C05487=1132.913,-86.314,-45.873,178.764,6.137,149.471
C05488=1132.907,-86.064,-45.883,178.766,6.138,149.470
C05489=1132.902,-85.815,-45.892,178.768,6.139,149.470
C05490=1132.896,-85.565,-45.902,178.770,6.139,149.469
C05491=1132.891,-85.315,-45.912,178.772,6.139,149.469
C05492=1132.886,-85.064,-45.921,178.774,6.140,149.468
C05493=1132.881,-84.815,-45.931,178.777,6.140,149.468
C05494=1132.875,-84.565,-45.940,178.778,6.140,149.467
C05495=1132.871,-84.316,-45.950,178.780,6.141,149.467
C05496=1132.865,-84.066,-45.960,178.783,6.142,149.466
C05497=1132.860,-83.816,-45.969,178.785,6.143,149.466
C05498=1132.854,-83.566,-45.979,178.786,6.143,149.465
C05499=1132.849,-83.317,-45.988,178.789,6.143,149.465
C05500=1132.843,-83.067,-45.998,178.791,6.144,149.464
C05501=1132.838,-82.818,-46.007,178.793,6.144,149.464
C05502=1132.833,-82.567,-46.018,178.795,6.144,149.463
C05503=1132.828,-82.318,-46.027,178.797,6.145,149.463
C05504=1132.822,-82.068,-46.037,178.799,6.146,149.462
C05505=1132.817,-81.818,-46.046,178.802,6.147,149.462
C05506=1132.812,-81.569,-46.056,178.804,6.146,149.461
C05507=1132.806,-81.318,-46.066,178.806,6.147,149.461
C05508=1132.801,-81.069,-46.075,178.808,6.148,149.460
C05509=1132.795,-80.820,-46.086,178.810,6.149,149.460
C05510=1132.791,-80.569,-46.095,178.812,6.148,149.459
C05511=1132.785,-80.320,-46.105,178.814,6.149,149.459
C05512=1132.779,-80.069,-46.114,178.816,6.150,149.458
C05513=1132.774,-79.820,-46.124,178.819,6.150,149.457
C05514=1132.769,-79.571,-46.134,178.821,6.150,149.457
C05515=1132.764,-79.321,-46.143,178.823,6.151,149.456
C05516=1132.758,-79.071,-46.153,178.825,6.152,149.456
C05517=1132.753,-78.821,-46.164,178.827,6.153,149.456
C05518=1132.748,-78.571,-46.173,178.829,6.153,149.455
C05519=1132.742,-78.322,-46.183,178.831,6.153,149.455
C05520=1132.737,-78.072,-46.193,178.834,6.154,149.454
C05521=1132.732,-77.822,-46.202,178.836,6.154,149.453
C05522=1132.726,-77.573,-46.212,178.837,6.154,149.453
C05523=1132.721,-77.301,-46.223,178.840,6.155,149.452
C05524=1132.715,-77.029,-46.234,178.842,6.156,149.452
C05525=1132.709,-76.759,-46.245,178.844,6.156,149.451
C05526=1132.703,-76.487,-46.255,178.847,6.157,149.451
C05527=1132.698,-76.237,-46.265,178.849,6.158,149.450
C05528=1132.693,-75.987,-46.276,178.852,6.158,149.450
C05529=1132.687,-75.737,-46.285,178.853,6.158,149.449
C05530=1132.682,-75.487,-46.295,178.855,6.159,149.449
C05531=1132.676,-75.238,-46.305,178.858,6.160,149.448
C05532=1132.671,-74.988,-46.315,178.860,6.160,149.448
C05533=1132.666,-74.738,-46.325,178.862,6.161,149.447
C05534=1132.661,-74.488,-46.335,178.864,6.161,149.446
C05535=1132.655,-74.239,-46.345,178.866,6.162,149.446
C05536=1132.649,-73.989,-46.355,178.868,6.162,149.445
C05537=1132.644,-73.739,-46.364,178.871,6.163,149.445
C05538=1132.639,-73.489,-46.375,178.872,6.163,149.444
C05539=1132.634,-73.240,-46.385,178.874,6.164,149.444
C05540=1132.628,-72.990,-46.395,178.877,6.164,149.443
C05541=1132.623,-72.741,-46.405,178.879,6.165,149.443
C05542=1132.618,-72.490,-46.415,178.881,6.166,149.442
C05543=1132.612,-72.240,-46.425,178.883,6.166,149.442
C05544=1132.607,-71.991,-46.435,178.885,6.166,149.441
C05545=1132.602,-71.742,-46.445,178.888,6.167,149.441
C05546=1132.597,-71.491,-46.455,178.890,6.167,149.440
C05547=1132.591,-71.242,-46.465,178.892,6.168,149.440
C05548=1132.586,-70.992,-46.476,178.894,6.168,149.439
C05549=1132.581,-70.743,-46.485,178.896,6.169,149.439
C05550=1132.576,-70.493,-46.496,178.898,6.170,149.438
C05551=1132.570,-70.243,-46.505,178.901,6.170,149.438
C05552=1132.564,-69.993,-46.515,178.903,6.171,149.437
C05553=1132.559,-69.743,-46.526,178.905,6.171,149.437
C05554=1132.554,-69.493,-46.536,178.907,6.172,149.436
C05555=1132.549,-69.244,-46.546,178.909,6.172,149.436
C05556=1132.543,-68.994,-46.556,178.912,6.173,149.435
C05557=1132.538,-68.744,-46.567,178.914,6.173,149.434
C05558=1132.533,-68.495,-46.577,178.916,6.174,149.434
C05559=1132.527,-68.245,-46.587,178.918,6.174,149.433
C05560=1132.522,-67.995,-46.598,178.920,6.175,149.433
C05561=1132.517,-67.746,-46.607,178.923,6.175,149.432
C05562=1132.511,-67.496,-46.617,178.925,6.176,149.432
C05563=1132.506,-67.246,-46.628,178.927,6.177,149.431
C05564=1132.501,-66.996,-46.638,178.929,6.177,149.431
C05565=1132.495,-66.747,-46.648,178.931,6.178,149.430
C05566=1132.490,-66.497,-46.659,178.933,6.178,149.430
C05567=1132.485,-66.247,-46.669,178.936,6.179,149.429
C05568=1132.480,-65.998,-46.679,178.938,6.180,149.429
C05569=1132.475,-65.748,-46.689,178.940,6.180,149.428
C05570=1132.469,-65.498,-46.700,178.942,6.180,149.428
C05571=1132.464,-65.248,-46.710,178.944,6.181,149.427
C05572=1132.459,-64.998,-46.720,178.946,6.181,149.426
C05573=1132.453,-64.749,-46.731,178.949,6.182,149.426
C05574=1132.447,-64.499,-46.741,178.951,6.183,149.426
C05575=1132.442,-64.249,-46.751,178.953,6.184,149.425
C05576=1132.437,-63.999,-46.762,178.955,6.184,149.425
C05577=1132.432,-63.749,-46.772,178.957,6.184,149.424
C05578=1132.426,-63.500,-46.782,178.959,6.185,149.423
C05579=1132.422,-63.251,-46.793,178.962,6.186,149.423
C05580=1132.417,-63.001,-46.803,178.964,6.186,149.422
C05581=1132.411,-62.751,-46.813,178.967,6.187,149.422
C05582=1132.406,-62.502,-46.824,178.969,6.187,149.421
C05583=1132.401,-62.251,-46.834,178.970,6.187,149.421
C05584=1132.395,-62.002,-46.844,178.973,6.188,149.420
C05585=1132.390,-61.752,-46.855,178.975,6.189,149.420
C05586=1132.385,-61.503,-46.866,178.977,6.189,149.419
C05587=1132.380,-61.252,-46.877,178.980,6.190,149.419
C05588=1132.374,-61.003,-46.887,178.982,6.191,149.418
C05589=1132.368,-60.753,-46.897,178.984,6.192,149.418
C05590=1132.363,-60.503,-46.908,178.986,6.192,149.417
C05591=1132.358,-60.254,-46.918,178.988,6.192,149.416
C05592=1132.353,-60.004,-46.929,178.990,6.193,149.416
C05593=1132.348,-59.754,-46.939,178.993,6.194,149.415
C05594=1132.343,-59.504,-46.950,178.995,6.194,149.415
C05595=1132.337,-59.255,-46.960,178.997,6.195,149.414
C05596=1132.331,-59.005,-46.970,179.000,6.195,149.414
C05597=1132.327,-58.755,-46.982,179.002,6.196,149.413
C05598=1132.321,-58.506,-46.992,179.003,6.196,149.413
C05599=1132.316,-58.256,-47.002,179.006,6.197,149.412
C05600=1132.310,-58.006,-47.013,179.008,6.197,149.412
C05601=1132.306,-57.756,-47.024,179.010,6.198,149.411
C05602=1132.300,-57.507,-47.034,179.013,6.199,149.411
C05603=1132.294,-57.256,-47.045,179.015,6.200,149.410
C05604=1132.289,-57.007,-47.056,179.018,6.200,149.410
C05605=1132.284,-56.757,-47.067,179.020,6.201,149.409
C05606=1132.279,-56.508,-47.077,179.021,6.201,149.409
C05607=1132.274,-56.258,-47.088,179.024,6.202,149.408
C05608=1132.268,-56.008,-47.098,179.026,6.202,149.408
C05609=1132.263,-55.758,-47.109,179.028,6.203,149.407
C05610=1132.258,-55.509,-47.120,179.031,6.203,149.406
C05611=1132.253,-55.259,-47.130,179.033,6.204,149.406
C05612=1132.247,-55.009,-47.141,179.035,6.205,149.405
C05613=1132.243,-54.760,-47.152,179.038,6.205,149.405
C05614=1132.237,-54.510,-47.162,179.040,6.206,149.404
C05615=1132.231,-54.260,-47.173,179.042,6.207,149.404
C05616=1132.226,-54.011,-47.184,179.044,6.207,149.403
C05617=1132.221,-53.761,-47.195,179.046,6.208,149.403
C05618=1132.215,-53.511,-47.205,179.048,6.208,149.402
C05619=1132.211,-53.261,-47.216,179.051,6.209,149.402
C05620=1132.205,-53.012,-47.227,179.053,6.210,149.401
C05621=1132.200,-52.762,-47.238,179.055,6.210,149.401
C05622=1132.194,-52.512,-47.249,179.058,6.211,149.400
C05623=1132.189,-52.263,-47.260,179.060,6.211,149.400
C05624=1132.184,-52.013,-47.270,179.062,6.212,149.399
C05625=1132.179,-51.763,-47.281,179.064,6.213,149.399
C05626=1132.174,-51.514,-47.292,179.067,6.213,149.398
C05627=1132.168,-51.243,-47.304,179.069,6.214,149.397
C05628=1132.162,-50.971,-47.315,179.071,6.215,149.397
C05629=1132.156,-50.701,-47.327,179.074,6.215,149.396
C05630=1132.151,-50.431,-47.339,179.076,6.216,149.396
C05631=1132.145,-50.180,-47.350,179.079,6.216,149.395
C05632=1132.140,-49.931,-47.361,179.081,6.217,149.395
C05633=1132.135,-49.681,-47.372,179.083,6.218,149.394
C05634=1132.130,-49.432,-47.383,179.085,6.219,149.394
C05635=1132.124,-49.181,-47.394,179.088,6.219,149.393
C05636=1132.119,-48.932,-47.405,179.090,6.219,149.392
C05637=1132.114,-48.683,-47.416,179.092,6.220,149.392
C05638=1132.109,-48.433,-47.427,179.094,6.221,149.391
C05639=1132.103,-48.183,-47.438,179.097,6.221,149.391
C05640=1132.098,-47.933,-47.449,179.099,6.222,149.390
C05641=1132.093,-47.684,-47.460,179.101,6.223,149.390
C05642=1132.088,-47.434,-47.470,179.103,6.223,149.389
C05643=1132.082,-47.184,-47.482,179.106,6.224,149.389
C05644=1132.077,-46.935,-47.493,179.108,6.225,149.388
C05645=1132.072,-46.685,-47.504,179.110,6.225,149.388
C05646=1132.066,-46.435,-47.515,179.113,6.226,149.387
C05647=1132.061,-46.185,-47.526,179.115,6.226,149.386
C05648=1132.056,-45.936,-47.537,179.117,6.227,149.386
C05649=1132.050,-45.686,-47.548,179.120,6.228,149.386
C05650=1132.045,-45.436,-47.559,179.122,6.229,149.385
C05651=1132.040,-45.187,-47.570,179.124,6.229,149.384
C05652=1132.034,-44.937,-47.582,179.127,6.230,149.384
C05653=1132.029,-44.687,-47.592,179.129,6.231,149.383
C05654=1132.025,-44.437,-47.604,179.131,6.231,149.383
C05655=1132.019,-44.188,-47.615,179.134,6.232,149.382
C05656=1132.014,-43.938,-47.626,179.135,6.232,149.382
C05657=1132.009,-43.688,-47.637,179.137,6.233,149.381
C05658=1132.003,-43.439,-47.649,179.140,6.233,149.381
C05659=1131.998,-43.189,-47.659,179.142,6.234,149.380
C05660=1131.993,-42.939,-47.671,179.144,6.235,149.380
C05661=1131.987,-42.690,-47.682,179.147,6.235,149.379
C05662=1131.983,-42.440,-47.693,179.149,6.236,149.379
C05663=1131.977,-42.190,-47.704,179.152,6.236,149.378
C05664=1131.972,-41.941,-47.715,179.154,6.237,149.377
C05665=1131.967,-41.691,-47.727,179.156,6.238,149.377
C05666=1131.961,-41.441,-47.739,179.159,6.238,149.376
C05667=1131.956,-41.191,-47.749,179.161,6.239,149.376
C05668=1131.950,-40.942,-47.761,179.163,6.240,149.375
C05669=1131.946,-40.692,-47.772,179.165,6.241,149.375
C05670=1131.940,-40.442,-47.784,179.168,6.241,149.374
C05671=1131.935,-40.193,-47.794,179.170,6.242,149.374
C05672=1131.929,-39.943,-47.806,179.172,6.243,149.373
C05673=1131.925,-39.693,-47.817,179.174,6.243,149.373
C05674=1131.920,-39.444,-47.828,179.177,6.244,149.372
C05675=1131.914,-39.194,-47.840,179.179,6.245,149.372
C05676=1131.909,-38.945,-47.851,179.181,6.245,149.371
C05677=1131.903,-38.694,-47.862,179.184,6.246,149.371
C05678=1131.898,-38.445,-47.873,179.186,6.247,149.370
C05679=1131.893,-38.195,-47.885,179.188,6.247,149.369
C05680=1131.888,-37.946,-47.897,179.191,6.248,149.369
C05681=1131.883,-37.696,-47.908,179.193,6.248,149.368
C05682=1131.877,-37.447,-47.919,179.195,6.249,149.368
C05683=1131.872,-37.197,-47.931,179.198,6.250,149.367
C05684=1131.867,-36.947,-47.943,179.200,6.251,149.367
C05685=1131.861,-36.697,-47.954,179.203,6.251,149.366
C05686=1131.856,-36.447,-47.966,179.205,6.252,149.366
C05687=1131.851,-36.198,-47.976,179.207,6.253,149.365
C05688=1131.845,-35.948,-47.988,179.209,6.254,149.365
C05689=1131.841,-35.698,-48.000,179.212,6.254,149.364
C05690=1131.835,-35.448,-48.012,179.214,6.255,149.363
C05691=1131.830,-35.199,-48.022,179.216,6.256,149.363
C05692=1131.824,-34.949,-48.034,179.219,6.256,149.362
C05693=1131.820,-34.700,-48.046,179.221,6.257,149.362
C05694=1131.814,-34.450,-48.058,179.223,6.257,149.361
C05695=1131.809,-34.200,-48.069,179.225,6.258,149.361
C05696=1131.804,-33.951,-48.080,179.228,6.259,149.360
C05697=1131.798,-33.701,-48.092,179.230,6.259,149.360
C05698=1131.793,-33.451,-48.104,179.232,6.260,149.359
C05699=1131.788,-33.202,-48.115,179.235,6.261,149.359
C05700=1131.783,-32.952,-48.127,179.237,6.261,149.358
C05701=1131.778,-32.702,-48.139,179.239,6.262,149.358
C05702=1131.772,-32.453,-48.150,179.242,6.263,149.357
C05703=1131.767,-32.203,-48.161,179.245,6.264,149.356
C05704=1131.762,-31.953,-48.173,179.247,6.265,149.356
C05705=1131.756,-31.703,-48.185,179.249,6.266,149.355
C05706=1131.752,-31.454,-48.196,179.251,6.266,149.355
C05707=1131.746,-31.204,-48.209,179.254,6.267,149.354
C05708=1131.741,-30.954,-48.221,179.256,6.268,149.354
C05709=1131.736,-30.705,-48.232,179.258,6.268,149.353
C05710=1131.730,-30.456,-48.244,179.261,6.269,149.353
C05711=1131.725,-30.206,-48.256,179.263,6.270,149.352
C05712=1131.720,-29.956,-48.267,179.266,6.270,149.352
C05713=1131.715,-29.706,-48.279,179.268,6.271,149.351
C05714=1131.709,-29.456,-48.291,179.270,6.272,149.351
C05715=1131.705,-29.207,-48.303,179.273,6.272,149.350
C05716=1131.700,-28.957,-48.315,179.275,6.273,149.350
C05717=1131.693,-28.708,-48.326,179.277,6.273,149.349
C05718=1131.689,-28.458,-48.337,179.280,6.274,149.348
C05719=1131.683,-28.208,-48.349,179.282,6.275,149.348
C05720=1131.678,-27.958,-48.361,179.284,6.275,149.347
C05721=1131.673,-27.709,-48.374,179.287,6.276,149.347
C05722=1131.668,-27.459,-48.385,179.289,6.278,149.346
C05723=1131.663,-27.210,-48.397,179.292,6.279,149.346
C05724=1131.657,-26.960,-48.409,179.294,6.279,149.345
C05725=1131.653,-26.711,-48.421,179.296,6.280,149.345
C05726=1131.647,-26.461,-48.433,179.299,6.281,149.344
C05727=1131.642,-26.211,-48.445,179.301,6.281,149.343
C05728=1131.637,-25.961,-48.456,179.303,6.282,149.343
C05729=1131.632,-25.712,-48.468,179.306,6.283,149.343
C05730=1131.627,-25.462,-48.480,179.308,6.283,149.342
C05731=1131.621,-25.192,-48.493,179.311,6.284,149.341
C05732=1131.615,-24.922,-48.507,179.313,6.285,149.341
C05733=1131.609,-24.652,-48.519,179.316,6.286,149.340
C05734=1131.604,-24.382,-48.532,179.318,6.286,149.340
C05735=1131.598,-24.132,-48.544,179.321,6.287,149.339
C05736=1131.594,-23.883,-48.556,179.323,6.288,149.339
C05737=1131.588,-23.633,-48.568,179.325,6.288,149.338
C05738=1131.583,-23.383,-48.580,179.328,6.290,149.337
C05739=1131.578,-23.133,-48.592,179.331,6.290,149.337
C05740=1131.572,-22.883,-48.604,179.333,6.291,149.336
C05741=1131.567,-22.633,-48.616,179.335,6.292,149.336
C05742=1131.562,-22.384,-48.629,179.338,6.292,149.335
C05743=1131.557,-22.135,-48.640,179.340,6.293,149.335
C05744=1131.552,-21.885,-48.652,179.342,6.294,149.334
C05745=1131.547,-21.635,-48.665,179.345,6.294,149.334
C05746=1131.541,-21.385,-48.676,179.347,6.295,149.333
C05747=1131.536,-21.136,-48.689,179.349,6.296,149.333
C05748=1131.531,-20.886,-48.701,179.352,6.297,149.332
C05749=1131.525,-20.636,-48.713,179.355,6.298,149.331
C05750=1131.520,-20.387,-48.725,179.357,6.299,149.331
C05751=1131.515,-20.137,-48.737,179.359,6.299,149.331
C05752=1131.510,-19.888,-48.749,179.362,6.300,149.330
C05753=1131.505,-19.638,-48.761,179.364,6.301,149.329
C05754=1131.500,-19.389,-48.774,179.366,6.301,149.329
C05755=1131.494,-19.139,-48.786,179.369,6.302,149.328
C05756=1131.489,-18.889,-48.798,179.371,6.303,149.328
C05757=1131.484,-18.639,-48.810,179.374,6.304,149.327
C05758=1131.479,-18.390,-48.823,179.376,6.305,149.327
C05759=1131.473,-18.140,-48.835,179.378,6.305,149.326
C05760=1131.468,-17.891,-48.847,179.381,6.306,149.326
C05761=1131.463,-17.641,-48.859,179.383,6.307,149.325
C05762=1131.457,-17.392,-48.872,179.385,6.307,149.324
C05763=1131.453,-17.141,-48.884,179.388,6.308,149.324
C05764=1131.447,-16.892,-48.897,179.390,6.310,149.324
C05765=1131.442,-16.642,-48.909,179.393,6.310,149.323
C05766=1131.437,-16.392,-48.921,179.395,6.311,149.322
C05767=1131.432,-16.143,-48.934,179.397,6.312,149.322
C05768=1131.426,-15.893,-48.946,179.400,6.312,149.321
C05769=1131.421,-15.644,-48.958,179.402,6.313,149.321
C05770=1131.416,-15.394,-48.970,179.404,6.314,149.320
C05771=1131.411,-15.145,-48.983,179.407,6.315,149.320
C05772=1131.406,-14.895,-48.995,179.410,6.316,149.319
C05773=1131.401,-14.645,-49.007,179.412,6.316,149.319
C05774=1131.396,-14.395,-49.020,179.414,6.317,149.318
C05775=1131.391,-14.146,-49.033,179.417,6.318,149.317
C05776=1131.385,-13.896,-49.045,179.419,6.318,149.317
C05777=1131.380,-13.647,-49.057,179.421,6.319,149.317
C05778=1131.375,-13.397,-49.070,179.425,6.320,149.316
C05779=1131.369,-13.148,-49.082,179.427,6.321,149.315
C05780=1131.364,-12.898,-49.094,179.429,6.322,149.315
C05781=1131.360,-12.648,-49.107,179.431,6.323,149.314
C05782=1131.354,-12.398,-49.119,179.434,6.323,149.314
C05783=1131.348,-12.149,-49.132,179.436,6.324,149.313
C05784=1131.343,-11.899,-49.145,179.439,6.326,149.313
C05785=1131.338,-11.650,-49.157,179.441,6.326,149.312
C05786=1131.333,-11.400,-49.169,179.444,6.327,149.312
C05787=1131.328,-11.150,-49.182,179.446,6.328,149.311
C05788=1131.323,-10.901,-49.195,179.448,6.328,149.310
C05789=1131.318,-10.651,-49.208,179.451,6.330,149.310
C05790=1131.313,-10.401,-49.219,179.453,6.330,149.310
C05791=1131.307,-10.152,-49.232,179.456,6.331,149.309
C05792=1131.302,-9.902,-49.246,179.458,6.332,149.308
C05793=1131.297,-9.652,-49.258,179.460,6.332,149.308
C05794=1131.292,-9.403,-49.271,179.463,6.333,149.307
C05795=1131.287,-9.153,-49.283,179.466,6.334,149.307
C05796=1131.281,-8.904,-49.295,179.468,6.335,149.306
C05797=1131.277,-8.654,-49.308,179.470,6.336,149.306
C05798=1131.271,-8.404,-49.321,179.473,6.336,149.305
C05799=1131.266,-8.155,-49.334,179.475,6.337,149.305
C05800=1131.261,-7.906,-49.347,179.478,6.339,149.304
C05801=1131.256,-7.655,-49.359,179.480,6.339,149.303
C05802=1131.251,-7.406,-49.371,179.483,6.340,149.303
C05803=1131.245,-7.156,-49.385,179.485,6.341,149.303
C05804=1131.240,-6.907,-49.397,179.487,6.341,149.302
C05805=1131.235,-6.657,-49.410,179.490,6.343,149.301
C05806=1131.230,-6.407,-49.423,179.492,6.344,149.301
C05807=1131.225,-6.158,-49.435,179.495,6.344,149.300
C05808=1131.219,-5.908,-49.449,179.497,6.345,149.300
C05809=1131.215,-5.658,-49.462,179.499,6.346,149.299
C05810=1131.210,-5.409,-49.474,179.502,6.347,149.299
C05811=1131.204,-5.160,-49.487,179.505,6.348,149.298
C05812=1131.199,-4.910,-49.500,179.507,6.348,149.298
C05813=1131.194,-4.660,-49.513,179.509,6.349,149.297
C05814=1131.189,-4.411,-49.526,179.512,6.350,149.296
C05815=1131.183,-4.161,-49.539,179.515,6.351,149.296
C05816=1131.179,-3.911,-49.552,179.517,6.352,149.296
C05817=1131.173,-3.662,-49.564,179.520,6.352,149.295
C05818=1131.168,-3.413,-49.577,179.522,6.353,149.294
C05819=1131.162,-3.163,-49.590,179.525,6.355,149.294
C05820=1131.158,-2.913,-49.603,179.527,6.355,149.293
C05821=1131.153,-2.664,-49.616,179.529,6.356,149.293
C05822=1131.147,-2.414,-49.629,179.532,6.357,149.292
C05823=1131.142,-2.164,-49.642,179.534,6.358,149.292
C05824=1131.137,-1.915,-49.654,179.537,6.359,149.291
C05825=1131.131,-1.665,-49.668,179.539,6.360,149.291
C05826=1131.127,-1.415,-49.681,179.541,6.360,149.290
C05827=1131.122,-1.166,-49.693,179.545,6.362,149.290
C05828=1131.116,-0.916,-49.706,179.547,6.362,149.289
C05829=1131.111,-0.666,-49.719,179.549,6.363,149.289
C05830=1131.106,-0.416,-49.733,179.552,6.364,149.288
C05831=1131.101,-0.168,-49.746,179.554,6.364,149.287
C05832=1131.096,0.082,-49.759,179.557,6.366,149.287
C05833=1131.090,0.332,-49.772,179.559,6.366,149.286
C05834=1131.085,0.581,-49.785,179.561,6.367,149.286
C05835=1131.079,0.851,-49.799,179.564,6.369,149.285
C05836=1131.075,1.120,-49.813,179.567,6.369,149.285
C05837=1131.068,1.390,-49.827,179.570,6.371,149.284
C05838=1131.063,1.660,-49.842,179.572,6.371,149.284
C05839=1131.058,1.910,-49.854,179.574,6.372,149.283
C05840=1131.053,2.159,-49.868,179.578,6.373,149.282
C05841=1131.047,2.408,-49.881,179.580,6.374,149.282
C05842=1131.043,2.658,-49.894,179.582,6.375,149.281
C05843=1131.037,2.908,-49.907,179.584,6.376,149.281
C05844=1131.033,3.158,-49.920,179.587,6.377,149.280
C05845=1131.027,3.407,-49.934,179.590,6.378,149.280
C05846=1131.022,3.656,-49.947,179.592,6.378,149.279
C05847=1131.017,3.906,-49.960,179.594,6.379,149.279
C05848=1131.012,4.155,-49.974,179.597,6.380,149.278
C05849=1131.007,4.406,-49.987,179.599,6.381,149.278
C05850=1131.001,4.655,-50.000,179.602,6.382,149.277
C05851=1130.996,4.905,-50.013,179.605,6.383,149.277
C05852=1130.991,5.154,-50.027,179.607,6.384,149.276
C05853=1130.985,5.403,-50.040,179.610,6.384,149.275
C05854=1130.981,5.653,-50.053,179.612,6.385,149.275
C05855=1130.975,5.902,-50.067,179.615,6.387,149.274
C05856=1130.971,6.153,-50.080,179.617,6.387,149.274
C05857=1130.965,6.402,-50.093,179.620,6.388,149.273
C05858=1130.960,6.652,-50.107,179.622,6.390,149.273
C05859=1130.955,6.901,-50.120,179.624,6.391,149.272
C05860=1130.950,7.151,-50.134,179.627,6.391,149.272
C05861=1130.945,7.400,-50.147,179.629,6.392,149.271
C05862=1130.940,7.651,-50.160,179.632,6.393,149.271
C05863=1130.935,7.899,-50.173,179.635,6.394,149.270
C05864=1130.930,8.150,-50.187,179.637,6.395,149.270
C05865=1130.924,8.399,-50.201,179.640,6.396,149.269
C05866=1130.919,8.649,-50.214,179.642,6.397,149.268
C05867=1130.914,8.898,-50.228,179.645,6.397,149.268
C05868=1130.909,9.148,-50.241,179.647,6.399,149.268
C05869=1130.904,9.397,-50.254,179.650,6.399,149.267
C05870=1130.899,9.647,-50.268,179.652,6.400,149.266
C05871=1130.893,9.896,-50.281,179.655,6.402,149.266
C05872=1130.888,10.146,-50.295,179.658,6.402,149.265
C05873=1130.883,10.396,-50.308,179.660,6.403,149.265
C05874=1130.878,10.645,-50.322,179.662,6.405,149.264
C05875=1130.873,10.895,-50.335,179.665,6.405,149.264
C05876=1130.868,11.144,-50.349,179.667,6.406,149.263
C05877=1130.862,11.394,-50.362,179.670,6.407,149.263
C05878=1130.858,11.643,-50.376,179.672,6.408,149.262
C05879=1130.853,11.893,-50.391,179.675,6.409,149.262
C05880=1130.847,12.142,-50.403,179.678,6.410,149.261
C05881=1130.842,12.392,-50.417,179.680,6.411,149.261
C05882=1130.837,12.642,-50.431,179.683,6.412,149.260
C05883=1130.832,12.891,-50.444,179.685,6.413,149.260
C05884=1130.827,13.141,-50.458,179.687,6.414,149.259
C05885=1130.822,13.390,-50.472,179.690,6.414,149.258
C05886=1130.817,13.640,-50.486,179.693,6.416,149.258
C05887=1130.811,13.890,-50.499,179.695,6.417,149.257
C05888=1130.807,14.139,-50.513,179.697,6.418,149.257
C05889=1130.801,14.388,-50.527,179.701,6.419,149.256
C05890=1130.796,14.639,-50.540,179.703,6.420,149.256
C05891=1130.792,14.888,-50.554,179.705,6.420,149.255
C05892=1130.786,15.137,-50.568,179.708,6.422,149.255
C05893=1130.781,15.387,-50.582,179.710,6.422,149.254
C05894=1130.775,15.636,-50.596,179.712,6.423,149.254
C05895=1130.771,15.886,-50.609,179.716,6.424,149.253
C05896=1130.766,16.136,-50.623,179.718,6.425,149.253
C05897=1130.760,16.385,-50.637,179.720,6.426,149.252
C05898=1130.755,16.635,-50.651,179.723,6.427,149.251
C05899=1130.750,16.884,-50.665,179.725,6.428,149.251
C05900=1130.745,17.134,-50.678,179.728,6.430,149.251
C05901=1130.740,17.384,-50.692,179.731,6.430,149.250
C05902=1130.735,17.633,-50.706,179.733,6.431,149.249
C05903=1130.730,17.882,-50.720,179.736,6.433,149.249
C05904=1130.724,18.133,-50.734,179.738,6.433,149.249
C05905=1130.719,18.382,-50.748,179.741,6.434,149.248
C05906=1130.715,18.631,-50.761,179.743,6.435,149.247
C05907=1130.710,18.881,-50.776,179.746,6.436,149.247
C05908=1130.704,19.130,-50.790,179.749,6.437,149.246
C05909=1130.699,19.380,-50.803,179.751,6.438,149.246
C05910=1130.694,19.630,-50.817,179.753,6.439,149.245
C05911=1130.689,19.879,-50.832,179.756,6.440,149.245
C05912=1130.683,20.128,-50.846,179.759,6.441,149.244
C05913=1130.678,20.378,-50.860,179.761,6.443,149.244
C05914=1130.673,20.628,-50.874,179.764,6.444,149.243
C05915=1130.669,20.877,-50.888,179.766,6.444,149.243
C05916=1130.663,21.127,-50.901,179.769,6.446,149.242
C05917=1130.658,21.377,-50.915,179.771,6.446,149.242
C05918=1130.653,21.626,-50.930,179.774,6.448,149.241
C05919=1130.648,21.875,-50.944,179.777,6.448,149.241
C05920=1130.643,22.125,-50.958,179.779,6.449,149.240
C05921=1130.638,22.375,-50.972,179.782,6.450,149.239
C05922=1130.632,22.624,-50.986,179.784,6.451,149.239
C05923=1130.627,22.873,-51.000,179.787,6.453,149.238
C05924=1130.623,23.123,-51.015,179.790,6.453,149.238
C05925=1130.618,23.373,-51.029,179.792,6.454,149.237
C05926=1130.612,23.622,-51.043,179.795,6.456,149.237
C05927=1130.607,23.872,-51.057,179.797,6.457,149.236
C05928=1130.602,24.121,-51.071,179.800,6.458,149.236
C05929=1130.597,24.371,-51.086,179.802,6.459,149.235
C05930=1130.592,24.621,-51.100,179.804,6.459,149.235
C05931=1130.587,24.870,-51.114,179.808,6.461,149.234
C05932=1130.582,25.119,-51.128,179.810,6.461,149.234
C05933=1130.577,25.369,-51.142,179.813,6.463,149.233
C05934=1130.572,25.619,-51.157,179.815,6.463,149.233
C05935=1130.566,25.868,-51.171,179.818,6.465,149.232
C05936=1130.561,26.118,-51.185,179.820,6.466,149.232
C05937=1130.556,26.367,-51.199,179.822,6.467,149.231
C05938=1130.551,26.617,-51.213,179.826,6.468,149.231
C05939=1130.546,26.886,-51.229,179.828,6.470,149.230
C05940=1130.540,27.155,-51.245,179.831,6.470,149.229
C05941=1130.534,27.424,-51.260,179.834,6.472,149.229
C05942=1130.529,27.692,-51.276,179.836,6.472,149.228
C05943=1130.524,27.942,-51.290,179.839,6.474,149.228
C05944=1130.519,28.192,-51.304,179.841,6.474,149.227
C05945=1130.514,28.442,-51.319,179.845,6.476,149.227
C05946=1130.509,28.691,-51.333,179.847,6.477,149.226
C05947=1130.504,28.941,-51.348,179.850,6.478,149.226
C05948=1130.498,29.190,-51.362,179.852,6.479,149.225
C05949=1130.493,29.439,-51.377,179.855,6.480,149.225
C05950=1130.489,29.689,-51.391,179.857,6.481,149.224
C05951=1130.484,29.939,-51.405,179.860,6.483,149.224
C05952=1130.479,30.188,-51.420,179.863,6.483,149.223
C05953=1130.474,30.438,-51.434,179.865,6.484,149.223
C05954=1130.468,30.688,-51.449,179.867,6.485,149.222
C05955=1130.463,30.937,-51.464,179.870,6.486,149.222
C05956=1130.458,31.186,-51.478,179.873,6.488,149.221
C05957=1130.453,31.435,-51.492,179.875,6.488,149.221
C05958=1130.448,31.685,-51.507,179.878,6.490,149.220
C05959=1130.442,31.935,-51.522,179.880,6.490,149.219
C05960=1130.438,32.184,-51.537,179.883,6.492,149.219
C05961=1130.433,32.434,-51.551,179.885,6.493,149.218
C05962=1130.428,32.684,-51.565,179.889,6.494,149.218
C05963=1130.423,32.933,-51.580,179.891,6.495,149.217
C05964=1130.418,33.183,-51.595,179.894,6.497,149.217
C05965=1130.413,33.433,-51.609,179.896,6.497,149.216
C05966=1130.408,33.682,-51.624,179.899,6.499,149.216
C05967=1130.402,33.931,-51.638,179.901,6.499,149.215
C05968=1130.397,34.181,-51.653,179.904,6.501,149.215
C05969=1130.392,34.430,-51.668,179.907,6.501,149.214
C05970=1130.387,34.679,-51.682,179.909,6.503,149.214
C05971=1130.382,34.929,-51.698,179.912,6.504,149.213
C05972=1130.377,35.179,-51.712,179.914,6.505,149.213
C05973=1130.372,35.428,-51.727,179.917,6.506,149.212
C05974=1130.367,35.677,-51.741,179.920,6.508,149.212
C05975=1130.361,35.927,-51.756,179.922,6.508,149.211
C05976=1130.357,36.176,-51.771,179.925,6.510,149.211
C05977=1130.352,36.426,-51.786,179.927,6.510,149.210
C05978=1130.346,36.676,-51.801,179.930,6.512,149.210
C05979=1130.342,36.925,-51.815,179.932,6.513,149.209
C05980=1130.337,37.174,-51.830,179.935,6.514,149.209
C05981=1130.331,37.424,-51.845,179.938,6.515,149.208
C05982=1130.327,37.673,-51.860,179.940,6.517,149.208
C05983=1130.321,37.924,-51.875,179.943,6.517,149.207
C05984=1130.316,38.173,-51.890,179.946,6.519,149.207
C05985=1130.311,38.422,-51.904,179.948,6.519,149.206
C05986=1130.306,38.672,-51.920,179.951,6.521,149.206
C05987=1130.301,38.905,-51.934,179.953,6.522,149.205
C05988=1130.297,39.137,-51.948,179.956,6.523,149.204
C05989=1130.293,39.369,-51.962,179.958,6.524,149.204
C05990=1130.268,40.531,-52.031,179.713,7.030,149.388
C05991=1130.263,40.781,-52.047,179.714,7.034,149.388
C05992=1130.259,41.031,-52.062,179.715,7.039,149.389
C05993=1130.253,41.281,-52.077,179.716,7.043,149.390
C05994=1130.249,41.530,-52.092,179.718,7.047,149.390
C05995=1130.243,41.779,-52.108,179.719,7.052,149.391
C05996=1130.239,42.028,-52.123,179.721,7.056,149.391
C05997=1130.233,42.278,-52.138,179.722,7.060,149.392
C05998=1130.227,42.528,-52.153,179.723,7.064,149.392
C05999=1130.223,42.777,-52.168,179.724,7.069,149.393
C06000=1130.218,43.027,-52.184,179.726,7.073,149.394
C06001=1130.213,43.276,-52.199,179.727,7.077,149.394
C06002=1130.208,43.525,-52.215,179.728,7.081,149.395
C06003=1130.203,43.774,-52.230,179.729,7.085,149.395
C06004=1130.198,44.025,-52.244,179.731,7.089,149.396
C06005=1130.192,44.274,-52.260,179.732,7.093,149.396
C06006=1130.188,44.524,-52.275,179.733,7.098,149.397
C06007=1130.183,44.773,-52.291,179.734,7.102,149.398
C06008=1130.177,45.023,-52.307,179.736,7.106,149.398
C06009=1130.173,45.272,-52.322,179.737,7.110,149.399
C06010=1130.167,45.521,-52.337,179.738,7.114,149.399
C06011=1130.163,45.771,-52.353,179.740,7.118,149.400
C06012=1130.158,46.020,-52.368,179.741,7.123,149.400
C06013=1130.153,46.270,-52.384,179.742,7.127,149.401
C06014=1130.148,46.519,-52.399,179.743,7.131,149.401
C06015=1130.143,46.769,-52.415,179.745,7.135,149.402
C06016=1130.138,47.018,-52.430,179.746,7.139,149.403
C06017=1130.132,47.268,-52.446,179.747,7.143,149.403
C06018=1130.128,47.517,-52.461,179.749,7.147,149.404
C06019=1130.124,47.735,-52.475,179.750,7.151,149.404
C06020=1130.119,47.953,-52.488,179.751,7.154,149.404
C06021=1130.115,48.170,-52.501,179.752,7.159,149.405
C06022=1130.110,48.388,-52.516,179.753,7.162,149.406
C06023=1130.105,48.606,-52.529,179.755,7.166,149.406
C06024=1130.101,48.824,-52.543,179.755,7.169,149.406
C06025=1130.097,49.042,-52.556,179.757,7.173,149.407
C06026=1130.093,49.259,-52.570,179.758,7.176,149.407
C06027=1130.088,49.509,-52.586,179.759,7.180,149.408
C06028=1130.083,49.758,-52.601,179.761,7.185,149.408
C06029=1130.078,50.008,-52.616,179.762,7.189,149.409
C06030=1130.073,50.258,-52.632,179.763,7.194,149.410
C06031=1130.068,50.507,-52.648,179.765,7.198,149.410
C06032=1130.062,50.756,-52.664,179.766,7.202,149.411
C06033=1130.058,51.006,-52.680,179.768,7.206,149.411
C06034=1130.053,51.255,-52.695,179.769,7.210,149.412
C06035=1130.048,51.504,-52.711,179.770,7.214,149.412
C06036=1130.043,51.755,-52.727,179.771,7.218,149.413
C06037=1130.038,52.004,-52.742,179.773,7.222,149.413
C06038=1130.032,52.253,-52.759,179.774,7.226,149.414
C06039=1130.028,52.503,-52.774,179.776,7.230,149.414
C06040=1130.023,52.752,-52.790,179.777,7.234,149.415
C06041=1130.018,53.001,-52.805,179.778,7.239,149.415
C06042=1130.013,53.251,-52.822,179.780,7.243,149.416
C06043=1130.008,53.500,-52.837,179.781,7.247,149.416
C06044=1130.002,53.750,-52.853,179.782,7.251,149.417
C06045=1129.998,53.999,-52.870,179.783,7.255,149.417
C06046=1129.992,54.249,-52.885,179.785,7.259,149.418
C06047=1129.987,54.498,-52.901,179.786,7.263,149.419
C06048=1129.983,54.747,-52.918,179.788,7.267,149.419
C06049=1129.977,54.997,-52.933,179.789,7.271,149.419
C06050=1129.973,55.247,-52.949,179.790,7.275,149.420
C06051=1129.968,55.495,-52.965,179.792,7.279,149.420
C06052=1129.963,55.745,-52.980,179.793,7.284,149.421
C06053=1129.958,55.995,-52.996,179.795,7.287,149.422
C06054=1129.953,56.244,-53.013,179.796,7.292,149.422
C06055=1129.948,56.494,-53.029,179.797,7.296,149.423
C06056=1129.943,56.743,-53.045,179.799,7.300,149.423
C06057=1129.938,56.993,-53.061,179.800,7.304,149.424
C06058=1129.933,57.241,-53.077,179.801,7.308,149.424
C06059=1129.928,57.491,-53.093,179.803,7.312,149.425
C06060=1129.923,57.741,-53.109,179.804,7.316,149.425
C06061=1129.918,57.990,-53.125,179.806,7.320,149.426
C06062=1129.913,58.240,-53.141,179.807,7.324,149.426
C06063=1129.908,58.489,-53.157,179.808,7.328,149.427
C06064=1129.903,58.739,-53.173,179.810,7.332,149.427
C06065=1129.897,58.988,-53.190,179.811,7.336,149.428
C06066=1129.893,59.238,-53.206,179.813,7.340,149.428
C06067=1129.888,59.487,-53.222,179.814,7.345,149.429
C06068=1129.883,59.736,-53.239,179.815,7.348,149.429
C06069=1129.878,59.986,-53.255,179.817,7.352,149.430
C06070=1129.873,60.235,-53.271,179.818,7.357,149.430
C06071=1129.868,60.484,-53.287,179.819,7.361,149.431
C06072=1129.863,60.734,-53.304,179.821,7.364,149.431
C06073=1129.858,60.983,-53.320,179.821,7.368,149.432
C06074=1129.853,61.233,-53.336,179.823,7.372,149.432
C06075=1129.848,61.447,-53.350,179.825,7.376,149.433
C06076=1129.845,61.663,-53.364,179.826,7.379,149.433
C06077=1129.840,61.879,-53.378,179.827,7.383,149.433
C06078=1129.836,62.094,-53.392,179.828,7.386,149.434
C06079=1129.831,62.308,-53.407,179.830,7.390,149.434
C06080=1129.828,62.523,-53.421,179.831,7.393,149.435
C06081=1129.823,62.739,-53.435,179.832,7.397,149.435
C06082=1129.819,62.954,-53.449,179.833,7.400,149.436
C06083=1129.814,63.203,-53.465,179.834,7.404,149.436
C06084=1129.809,63.453,-53.482,179.836,7.408,149.437
C06085=1129.804,63.702,-53.499,179.837,7.412,149.437
C06086=1129.799,63.952,-53.514,179.838,7.416,149.438
C06087=1129.794,64.200,-53.531,179.840,7.420,149.438
C06088=1129.789,64.450,-53.547,179.842,7.424,149.439
C06089=1129.784,64.700,-53.565,179.843,7.428,149.439
C06090=1129.779,64.949,-53.580,179.844,7.432,149.440
C06091=1129.774,65.199,-53.597,179.846,7.436,149.440
C06092=1129.769,65.447,-53.613,179.847,7.440,149.441
C06093=1129.764,65.697,-53.631,179.848,7.445,149.441
C06094=1129.760,65.947,-53.647,179.850,7.448,149.442
C06095=1129.754,66.196,-53.663,179.852,7.452,149.442
C06096=1129.750,66.446,-53.679,179.853,7.457,149.443
C06097=1129.744,66.695,-53.697,179.854,7.461,149.443
C06098=1129.739,66.944,-53.713,179.856,7.464,149.443
C06099=1129.735,67.194,-53.730,179.857,7.468,149.444
C06100=1129.730,67.443,-53.747,179.859,7.473,149.445
C06101=1129.725,67.692,-53.763,179.860,7.477,149.445
C06102=1129.720,67.942,-53.780,179.862,7.480,149.445
C06103=1129.715,68.192,-53.797,179.863,7.485,149.446
C06104=1129.710,68.440,-53.813,179.864,7.489,149.446
C06105=1129.705,68.690,-53.830,179.866,7.493,149.447
C06106=1129.700,68.940,-53.847,179.868,7.496,149.447
C06107=1129.695,69.189,-53.863,179.868,7.500,149.448
C06108=1129.690,69.438,-53.880,179.870,7.504,149.448
C06109=1129.685,69.688,-53.897,179.871,7.508,149.449
C06110=1129.680,69.937,-53.913,179.873,7.512,149.449
C06111=1129.676,70.186,-53.931,179.874,7.516,149.450
C06112=1129.671,70.436,-53.948,179.875,7.520,149.450
C06113=1129.665,70.684,-53.964,179.877,7.524,149.451
C06114=1129.660,70.934,-53.981,179.878,7.528,149.451
C06115=1129.656,71.184,-53.998,179.880,7.532,149.452
C06116=1129.651,71.434,-54.015,179.881,7.536,149.452
C06117=1129.645,71.682,-54.032,179.883,7.540,149.453
C06118=1129.641,71.932,-54.048,179.884,7.544,149.453
C06119=1129.636,72.182,-54.066,179.886,7.548,149.454
C06120=1129.631,72.431,-54.082,179.887,7.552,149.454
C06121=1129.625,72.680,-54.099,179.889,7.556,149.455
C06122=1129.621,72.930,-54.116,179.890,7.560,149.455
C06123=1129.616,73.179,-54.134,179.891,7.564,149.456
C06124=1129.612,73.428,-54.151,179.893,7.568,149.456
C06125=1129.606,73.677,-54.167,179.895,7.572,149.457
C06126=1129.601,73.927,-54.184,179.896,7.576,149.457
C06127=1129.596,74.177,-54.201,179.897,7.580,149.458
C06128=1129.592,74.426,-54.219,179.899,7.584,149.458
C06129=1129.587,74.675,-54.236,179.900,7.588,149.458
C06130=1129.582,74.924,-54.252,179.902,7.592,149.459
C06131=1129.577,75.140,-54.267,179.903,7.595,149.459
C06132=1129.573,75.354,-54.282,179.905,7.599,149.460
C06133=1129.569,75.570,-54.297,179.905,7.602,149.460
C06134=1129.564,75.785,-54.312,179.907,7.606,149.461
C06135=1129.560,76.000,-54.327,179.908,7.609,149.461
C06136=1129.556,76.215,-54.341,179.910,7.613,149.461
C06137=1129.552,76.430,-54.356,179.911,7.616,149.462
C06138=1129.548,76.645,-54.371,179.912,7.619,149.462
C06139=1129.543,76.895,-54.388,179.913,7.623,149.463
C06140=1129.538,77.144,-54.405,179.914,7.626,149.463
C06141=1129.533,77.393,-54.423,179.915,7.631,149.464
C06142=1129.527,77.642,-54.440,179.916,7.634,149.464
C06143=1129.523,77.892,-54.457,179.917,7.638,149.465
C06144=1129.518,78.141,-54.475,179.918,7.641,149.465
C06145=1129.513,78.390,-54.491,179.919,7.645,149.466
C06146=1129.508,78.640,-54.509,179.920,7.649,149.467
C06147=1129.503,78.889,-54.527,179.921,7.653,149.467
C06148=1129.498,79.138,-54.543,179.922,7.656,149.468
C06149=1129.493,79.387,-54.561,179.923,7.660,149.468
C06150=1129.488,79.637,-54.578,179.924,7.663,149.469
C06151=1129.484,79.887,-54.595,179.925,7.668,149.469
C06152=1129.479,80.136,-54.613,179.926,7.671,149.470
C06153=1129.474,80.386,-54.630,179.927,7.675,149.470
C06154=1129.469,80.635,-54.647,179.928,7.678,149.471
C06155=1129.464,80.884,-54.665,179.929,7.682,149.471
C06156=1129.459,81.133,-54.683,179.931,7.686,149.472
C06157=1129.453,81.383,-54.700,179.931,7.690,149.473
C06158=1129.449,81.631,-54.717,179.933,7.694,149.473
C06159=1129.444,81.881,-54.734,179.934,7.697,149.474
C06160=1129.439,82.130,-54.752,179.935,7.701,149.474
C06161=1129.434,82.380,-54.769,179.936,7.705,149.475
C06162=1129.430,82.629,-54.787,179.937,7.709,149.475
C06163=1129.424,82.879,-54.804,179.938,7.713,149.476
C06164=1129.420,83.128,-54.822,179.940,7.717,149.476
C06165=1129.414,83.378,-54.839,179.941,7.720,149.477
C06166=1129.410,83.627,-54.857,179.942,7.724,149.477
C06167=1129.405,83.876,-54.875,179.944,7.728,149.478
C06168=1129.400,84.126,-54.892,179.945,7.732,149.478
C06169=1129.395,84.375,-54.910,179.946,7.735,149.479
C06170=1129.391,84.624,-54.927,179.947,7.739,149.479
C06171=1129.386,84.874,-54.945,179.948,7.744,149.480
C06172=1129.381,85.123,-54.963,179.950,7.748,149.480
C06173=1129.376,85.372,-54.980,179.951,7.751,149.481
C06174=1129.371,85.622,-54.998,179.953,7.755,149.481
C06175=1129.366,85.871,-55.016,179.954,7.759,149.482
C06176=1129.361,86.120,-55.032,179.955,7.763,149.482
C06177=1129.356,86.370,-55.050,179.957,7.767,149.483
C06178=1129.352,86.619,-55.068,179.957,7.770,149.483
C06179=1129.346,86.868,-55.086,179.959,7.774,149.484
C06180=1129.341,87.118,-55.104,179.961,7.778,149.484
C06181=1129.336,87.367,-55.122,179.962,7.782,149.484
C06182=1129.332,87.616,-55.140,179.963,7.786,149.485
C06183=1129.326,87.866,-55.157,179.965,7.790,149.486
C06184=1129.321,88.115,-55.175,179.967,7.794,149.486
C06185=1129.317,88.364,-55.192,179.968,7.798,149.486
C06186=1129.312,88.613,-55.210,179.969,7.801,149.487
C06187=1129.308,88.828,-55.225,179.971,7.805,149.487
C06188=1129.303,89.043,-55.241,179.972,7.808,149.488
C06189=1129.299,89.258,-55.256,179.973,7.812,149.488
C06190=1129.295,89.473,-55.272,179.974,7.815,149.489
C06191=1129.291,89.688,-55.287,179.975,7.818,149.489
C06192=1129.287,89.903,-55.303,179.977,7.822,149.489
C06193=1129.283,90.118,-55.317,179.978,7.825,149.490
C06194=1129.278,90.333,-55.333,179.980,7.828,149.490
C06195=1129.273,90.583,-55.351,179.981,7.832,149.490
C06196=1129.268,90.832,-55.369,179.983,7.836,149.491
C06197=1129.264,91.081,-55.387,179.985,7.840,149.491
C06198=1129.258,91.330,-55.405,179.986,7.844,149.492
C06199=1129.253,91.579,-55.423,179.988,7.848,149.492
C06200=1129.249,91.829,-55.442,179.989,7.852,149.493
C06201=1129.244,92.078,-55.460,179.991,7.856,149.493
C06202=1129.239,92.328,-55.478,179.992,7.860,149.494
C06203=1129.234,92.577,-55.496,179.994,7.864,149.494
C06204=1129.229,92.826,-55.514,179.995,7.868,149.495
C06205=1129.224,93.075,-55.532,179.997,7.872,149.495
C06206=1129.219,93.324,-55.550,179.999,7.875,149.495
C06207=1129.215,93.574,-55.568,-179.999,7.879,149.496
C06208=1129.210,93.823,-55.586,-179.998,7.883,149.496
C06209=1129.205,94.072,-55.604,-179.996,7.888,149.496
C06210=1129.200,94.322,-55.622,-179.994,7.892,149.497
C06211=1129.196,94.571,-55.640,-179.992,7.895,149.497
C06212=1129.191,94.820,-55.658,-179.991,7.899,149.498
C06213=1129.186,95.070,-55.677,-179.989,7.903,149.498
C06214=1129.181,95.319,-55.695,-179.988,7.907,149.499
C06215=1129.176,95.569,-55.713,-179.985,7.911,149.499
C06216=1129.171,95.818,-55.731,-179.983,7.915,149.499
C06217=1129.166,96.067,-55.749,-179.982,7.919,149.500
C06218=1129.162,96.317,-55.767,-179.980,7.923,149.500
C06219=1129.157,96.565,-55.786,-179.978,7.927,149.500
C06220=1129.151,96.815,-55.804,-179.976,7.931,149.501
C06221=1129.146,97.064,-55.822,-179.974,7.935,149.501
C06222=1129.142,97.313,-55.840,-179.973,7.939,149.502
C06223=1129.137,97.563,-55.859,-179.971,7.943,149.502
C06224=1129.133,97.812,-55.877,-179.968,7.947,149.502
C06225=1129.127,98.061,-55.896,-179.967,7.951,149.503
C06226=1129.122,98.310,-55.914,-179.965,7.955,149.503
C06227=1129.118,98.560,-55.932,-179.963,7.958,149.503
C06228=1129.113,98.809,-55.951,-179.961,7.963,149.504
C06229=1129.107,99.058,-55.969,-179.959,7.967,149.504
C06230=1129.103,99.307,-55.987,-179.957,7.971,149.504
C06231=1129.098,99.557,-56.006,-179.955,7.975,149.505
C06232=1129.094,99.806,-56.024,-179.953,7.979,149.505
C06233=1129.088,100.055,-56.043,-179.951,7.983,149.505
C06234=1129.084,100.305,-56.061,-179.949,7.987,149.506
C06235=1129.079,100.554,-56.080,-179.947,7.991,149.506
C06236=1129.073,100.803,-56.099,-179.945,7.995,149.506
C06237=1129.069,101.052,-56.118,-179.943,7.999,149.507
C06238=1129.065,101.302,-56.136,-179.941,8.003,149.507
C06239=1129.059,101.551,-56.154,-179.939,8.006,149.507
C06240=1129.055,101.800,-56.173,-179.937,8.011,149.508
C06241=1129.050,102.050,-56.191,-179.935,8.014,149.508
C06242=1129.045,102.298,-56.211,-179.932,8.019,149.508
C06243=1129.041,102.514,-56.226,-179.931,8.022,149.509
C06244=1129.037,102.728,-56.243,-179.929,8.025,149.509
C06245=1129.032,102.943,-56.258,-179.927,8.029,149.509
C06246=1129.028,103.159,-56.275,-179.925,8.032,149.509
C06247=1129.024,103.373,-56.291,-179.923,8.036,149.510
C06248=1129.019,103.588,-56.307,-179.921,8.040,149.510
C06249=1129.016,103.803,-56.323,-179.920,8.042,149.510
C06250=1129.011,104.018,-56.339,-179.918,8.046,149.510
C06251=1129.007,104.266,-56.358,-179.915,8.050,149.511
C06252=1129.002,104.516,-56.377,-179.913,8.054,149.511
C06253=1128.997,104.765,-56.396,-179.911,8.058,149.511
C06254=1128.992,105.015,-56.415,-179.909,8.062,149.511
C06255=1128.987,105.264,-56.433,-179.906,8.066,149.512
C06256=1128.982,105.513,-56.453,-179.904,8.070,149.512
C06257=1128.978,105.762,-56.471,-179.901,8.074,149.512
C06258=1128.972,106.011,-56.490,-179.900,8.078,149.513
C06259=1128.968,106.261,-56.509,-179.897,8.082,149.513
C06260=1128.963,106.510,-56.528,-179.895,8.086,149.513
C06261=1128.959,106.759,-56.547,-179.892,8.090,149.513
C06262=1128.953,107.008,-56.566,-179.890,8.093,149.513
C06263=1128.949,107.258,-56.585,-179.888,8.098,149.514
C06264=1128.944,107.507,-56.604,-179.885,8.102,149.514
C06265=1128.939,107.757,-56.624,-179.883,8.106,149.514
C06266=1128.934,108.005,-56.642,-179.880,8.110,149.514
C06267=1128.929,108.255,-56.661,-179.878,8.113,149.515
C06268=1128.925,108.504,-56.680,-179.875,8.118,149.515
C06269=1128.920,108.753,-56.699,-179.873,8.122,149.515
C06270=1128.915,109.002,-56.719,-179.871,8.125,149.515
C06271=1128.911,109.252,-56.738,-179.868,8.130,149.515
C06272=1128.905,109.500,-56.757,-179.866,8.133,149.516
C06273=1128.900,109.751,-56.776,-179.863,8.137,149.516
C06274=1128.896,109.999,-56.795,-179.860,8.142,149.516
C06275=1128.891,110.249,-56.814,-179.858,8.145,149.516
C06276=1128.886,110.498,-56.834,-179.855,8.149,149.516
C06277=1128.882,110.747,-56.853,-179.853,8.153,149.516
C06278=1128.876,110.996,-56.872,-179.851,8.157,149.517
C06279=1128.871,111.245,-56.892,-179.848,8.160,149.517
C06280=1128.867,111.494,-56.910,-179.847,8.164,149.517
C06281=1128.862,111.743,-56.930,-179.845,8.168,149.518
C06282=1128.857,111.993,-56.950,-179.843,8.171,149.518
C06283=1128.852,112.242,-56.969,-179.841,8.175,149.518
C06284=1128.848,112.491,-56.988,-179.839,8.178,149.518
C06285=1128.843,112.740,-57.007,-179.837,8.182,149.519
C06286=1128.838,112.990,-57.027,-179.835,8.186,149.519
C06287=1128.833,113.239,-57.047,-179.833,8.189,149.519
C06288=1128.829,113.488,-57.065,-179.831,8.193,149.519
C06289=1128.824,113.737,-57.085,-179.829,8.196,149.520
C06290=1128.819,113.986,-57.104,-179.827,8.200,149.520
C06291=1128.814,114.236,-57.124,-179.825,8.204,149.520
C06292=1128.809,114.485,-57.144,-179.823,8.207,149.520
C06293=1128.804,114.734,-57.163,-179.822,8.210,149.521
C06294=1128.800,114.983,-57.182,-179.820,8.213,149.521
C06295=1128.795,115.233,-57.202,-179.818,8.217,149.521
C06296=1128.790,115.481,-57.222,-179.816,8.221,149.522
C06297=1128.785,115.731,-57.241,-179.814,8.224,149.522
C06298=1128.780,115.980,-57.261,-179.812,8.228,149.522
C06299=1128.776,116.195,-57.278,-179.810,8.230,149.522
C06300=1128.772,116.410,-57.295,-179.808,8.234,149.522
C06301=1128.768,116.624,-57.311,-179.807,8.237,149.523
C06302=1128.764,116.839,-57.328,-179.805,8.239,149.523
C06303=1128.760,117.053,-57.345,-179.803,8.243,149.523
C06304=1128.756,117.269,-57.362,-179.802,8.245,149.523
C06305=1128.752,117.484,-57.379,-179.800,8.248,149.523
C06306=1128.747,117.698,-57.396,-179.798,8.252,149.524
C06307=1128.743,117.947,-57.416,-179.797,8.255,149.524
C06308=1128.738,118.197,-57.435,-179.795,8.258,149.524
C06309=1128.733,118.446,-57.455,-179.793,8.262,149.525
C06310=1128.728,118.694,-57.475,-179.791,8.265,149.525
C06311=1128.723,118.944,-57.495,-179.789,8.269,149.525
C06312=1128.719,119.194,-57.514,-179.787,8.273,149.525
C06313=1128.714,119.442,-57.534,-179.786,8.275,149.526
C06314=1128.709,119.691,-57.554,-179.784,8.279,149.526
C06315=1128.704,119.941,-57.574,-179.782,8.282,149.526
C06316=1128.700,120.190,-57.594,-179.780,8.286,149.526
C06317=1128.694,120.439,-57.613,-179.778,8.289,149.527
C06318=1128.690,120.688,-57.633,-179.777,8.292,149.527
C06319=1128.685,120.937,-57.653,-179.775,8.296,149.527
C06320=1128.680,121.187,-57.673,-179.773,8.299,149.527
C06321=1128.675,121.435,-57.693,-179.771,8.303,149.528
C06322=1128.671,121.685,-57.713,-179.768,8.306,149.528
C06323=1128.666,121.934,-57.732,-179.767,8.310,149.528
C06324=1128.661,122.183,-57.753,-179.765,8.313,149.529
C06325=1128.657,122.433,-57.772,-179.763,8.317,149.529
C06326=1128.652,122.681,-57.792,-179.761,8.320,149.529
C06327=1128.647,122.931,-57.812,-179.760,8.323,149.529
C06328=1128.642,123.180,-57.832,-179.758,8.327,149.530
C06329=1128.638,123.429,-57.852,-179.756,8.330,149.530
C06330=1128.633,123.678,-57.872,-179.754,8.334,149.530
C06331=1128.628,123.927,-57.892,-179.753,8.336,149.530
C06332=1128.623,124.176,-57.913,-179.751,8.340,149.531
C06333=1128.618,124.425,-57.933,-179.749,8.344,149.531
C06334=1128.614,124.675,-57.953,-179.748,8.346,149.531
C06335=1128.609,124.924,-57.973,-179.745,8.350,149.531
C06336=1128.604,125.173,-57.993,-179.743,8.353,149.532
C06337=1128.600,125.422,-58.013,-179.742,8.357,149.532
C06338=1128.595,125.671,-58.032,-179.740,8.360,149.532
C06339=1128.590,125.920,-58.053,-179.738,8.363,149.533
C06340=1128.585,126.169,-58.074,-179.736,8.367,149.533
C06341=1128.580,126.419,-58.093,-179.735,8.370,149.533
C06342=1128.576,126.668,-58.114,-179.733,8.374,149.533
C06343=1128.571,126.917,-58.134,-179.731,8.377,149.534
C06344=1128.567,127.166,-58.154,-179.730,8.380,149.534
C06345=1128.562,127.416,-58.175,-179.728,8.384,149.534
C06346=1128.557,127.665,-58.195,-179.726,8.387,149.534
C06347=1128.552,127.913,-58.214,-179.724,8.390,149.535
C06348=1128.547,128.162,-58.235,-179.722,8.393,149.535
C06349=1128.542,128.412,-58.256,-179.721,8.397,149.535
C06350=1128.538,128.661,-58.276,-179.719,8.400,149.536
C06351=1128.533,128.910,-58.296,-179.717,8.403,149.536
C06352=1128.528,129.159,-58.316,-179.715,8.407,149.536
C06353=1128.523,129.408,-58.337,-179.714,8.410,149.536
C06354=1128.519,129.657,-58.358,-179.712,8.414,149.537
C06355=1128.515,129.872,-58.375,-179.711,8.416,149.537
C06356=1128.511,130.086,-58.392,-179.709,8.419,149.537
C06357=1128.506,130.302,-58.410,-179.708,8.422,149.537
C06358=1128.502,130.516,-58.427,-179.706,8.424,149.538
C06359=1128.499,130.731,-58.445,-179.705,8.427,149.538
C06360=1128.495,130.946,-58.462,-179.703,8.431,149.538
C06361=1128.490,131.160,-58.480,-179.702,8.434,149.538
C06362=1128.486,131.374,-58.498,-179.700,8.436,149.539
C06363=1128.482,131.623,-58.518,-179.699,8.439,149.539
C06364=1128.476,131.873,-58.539,-179.697,8.443,149.539
C06365=1128.472,132.122,-58.559,-179.695,8.446,149.540
C06366=1128.467,132.371,-58.579,-179.694,8.449,149.540
C06367=1128.462,132.620,-58.600,-179.692,8.453,149.540
C06368=1128.458,132.869,-58.621,-179.691,8.456,149.540
C06369=1128.452,133.119,-58.642,-179.689,8.459,149.541
C06370=1128.448,133.367,-58.662,-179.688,8.462,149.541
C06371=1128.444,133.616,-58.682,-179.686,8.466,149.541
C06372=1128.438,133.866,-58.703,-179.683,8.469,149.542
C06373=1128.434,134.115,-58.724,-179.682,8.472,149.542
C06374=1128.429,134.364,-58.745,-179.680,8.476,149.542
C06375=1128.424,134.613,-58.765,-179.679,8.479,149.542
C06376=1128.420,134.862,-58.786,-179.677,8.483,149.543
C06377=1128.415,135.111,-58.807,-179.676,8.485,149.543
C06378=1128.410,135.360,-58.827,-179.674,8.489,149.544
C06379=1128.405,135.609,-58.848,-179.673,8.492,149.544
C06380=1128.401,135.858,-58.868,-179.671,8.495,149.544
C06381=1128.396,136.107,-58.889,-179.669,8.499,149.544
C06382=1128.391,136.356,-58.910,-179.668,8.502,149.545
C06383=1128.386,136.606,-58.931,-179.666,8.506,149.545
C06384=1128.382,136.855,-58.951,-179.665,8.508,149.545
C06385=1128.377,137.105,-58.972,-179.662,8.512,149.546
C06386=1128.372,137.354,-58.993,-179.661,8.515,149.546
C06387=1128.368,137.602,-59.014,-179.659,8.519,149.546
C06388=1128.363,137.851,-59.035,-179.658,8.522,149.547
C06389=1128.358,138.100,-59.056,-179.656,8.525,149.547
C06390=1128.354,138.349,-59.076,-179.655,8.528,149.547
C06391=1128.348,138.599,-59.097,-179.653,8.532,149.547
C06392=1128.344,138.848,-59.117,-179.652,8.535,149.548
C06393=1128.339,139.097,-59.138,-179.650,8.538,149.548
C06394=1128.335,139.345,-59.159,-179.649,8.541,149.549
C06395=1128.330,139.595,-59.181,-179.647,8.545,149.549
C06396=1128.326,139.844,-59.201,-179.646,8.548,149.549
C06397=1128.320,140.093,-59.222,-179.644,8.551,149.549
C06398=1128.316,140.342,-59.244,-179.643,8.555,149.550
C06399=1128.311,140.591,-59.264,-179.641,8.558,149.550
C06400=1128.306,140.840,-59.285,-179.640,8.561,149.551
C06401=1128.302,141.089,-59.305,-179.638,8.565,149.551
C06402=1128.297,141.338,-59.328,-179.637,8.568,149.551
C06403=1128.293,141.587,-59.348,-179.635,8.572,149.552
C06404=1128.288,141.837,-59.369,-179.634,8.574,149.552
C06405=1128.282,142.086,-59.390,-179.633,8.577,149.552
C06406=1128.278,142.334,-59.411,-179.631,8.581,149.553
C06407=1128.273,142.584,-59.432,-179.630,8.584,149.553
C06408=1128.269,142.833,-59.453,-179.628,8.587,149.553
C06409=1128.264,143.082,-59.474,-179.626,8.591,149.554
C06410=1128.259,143.331,-59.495,-179.625,8.594,149.554
C06411=1128.256,143.546,-59.513,-179.623,8.597,149.554
C06412=1128.251,143.760,-59.531,-179.622,8.600,149.555
C06413=1128.247,143.975,-59.550,-179.621,8.603,149.555
C06414=1128.244,144.189,-59.568,-179.619,8.606,149.555
C06415=1128.239,144.404,-59.587,-179.618,8.609,149.556
C06416=1128.235,144.618,-59.604,-179.617,8.611,149.556
C06417=1128.231,144.833,-59.623,-179.616,8.615,149.556
C06418=1128.227,145.048,-59.641,-179.615,8.616,149.556
C06419=1128.223,145.296,-59.662,-179.612,8.621,149.557
C06420=1128.217,145.546,-59.683,-179.610,8.625,149.557
C06421=1128.213,145.794,-59.705,-179.607,8.629,149.557
C06422=1128.209,146.044,-59.726,-179.604,8.633,149.557
C06423=1128.204,146.293,-59.747,-179.602,8.637,149.557
C06424=1128.199,146.542,-59.768,-179.599,8.641,149.558
C06425=1128.194,146.790,-59.790,-179.596,8.645,149.558
C06426=1128.189,147.040,-59.811,-179.593,8.649,149.558
C06427=1128.185,147.289,-59.832,-179.591,8.653,149.558
C06428=1128.180,147.538,-59.853,-179.588,8.657,149.558
C06429=1128.175,147.787,-59.875,-179.585,8.661,149.558
C06430=1128.170,148.037,-59.896,-179.583,8.664,149.559
C06431=1128.166,148.285,-59.918,-179.581,8.668,149.559
C06432=1128.161,148.534,-59.940,-179.577,8.672,149.559
C06433=1128.157,148.783,-59.960,-179.575,8.676,149.559
C06434=1128.152,149.032,-59.982,-179.573,8.680,149.559
C06435=1128.147,149.281,-60.004,-179.570,8.683,149.559
C06436=1128.143,149.531,-60.025,-179.567,8.687,149.560
C06437=1128.138,149.779,-60.047,-179.564,8.691,149.560
C06438=1128.133,150.028,-60.069,-179.562,8.695,149.560
C06439=1128.128,150.278,-60.090,-179.559,8.699,149.560
C06440=1128.123,150.527,-60.112,-179.557,8.702,149.560
C06441=1128.119,150.775,-60.133,-179.554,8.706,149.560
C06442=1128.114,151.025,-60.155,-179.552,8.710,149.560
C06443=1128.109,151.273,-60.177,-179.549,8.714,149.561
C06444=1128.104,151.522,-60.198,-179.546,8.717,149.561
C06445=1128.101,151.772,-60.219,-179.544,8.721,149.561
C06446=1128.096,152.020,-60.241,-179.541,8.724,149.561
C06447=1128.092,152.270,-60.263,-179.538,8.729,149.561
C06448=1128.087,152.518,-60.285,-179.536,8.732,149.561
C06449=1128.081,152.767,-60.307,-179.533,8.736,149.561
C06450=1128.076,153.017,-60.328,-179.531,8.739,149.561
C06451=1128.072,153.266,-60.350,-179.528,8.743,149.562
C06452=1128.067,153.515,-60.372,-179.525,8.746,149.562
C06453=1128.062,153.764,-60.394,-179.523,8.751,149.562
C06454=1128.058,154.012,-60.415,-179.520,8.754,149.562
C06455=1128.053,154.262,-60.438,-179.518,8.757,149.562
C06456=1128.048,154.510,-60.459,-179.515,8.761,149.562
C06457=1128.044,154.760,-60.481,-179.513,8.765,149.563
C06458=1128.039,155.008,-60.503,-179.510,8.769,149.563
C06459=1128.035,155.258,-60.525,-179.508,8.772,149.563
C06460=1128.030,155.506,-60.547,-179.505,8.775,149.563
C06461=1128.026,155.756,-60.569,-179.502,8.779,149.563
C06462=1128.020,156.005,-60.591,-179.500,8.783,149.563
C06463=1128.016,156.254,-60.613,-179.497,8.786,149.563
C06464=1128.011,156.503,-60.635,-179.495,8.790,149.563
C06465=1128.007,156.752,-60.657,-179.492,8.793,149.563
C06466=1128.002,157.001,-60.678,-179.490,8.796,149.563
C06467=1127.998,157.215,-60.698,-179.488,8.800,149.564
C06468=1127.994,157.430,-60.717,-179.485,8.803,149.564
C06469=1127.990,157.644,-60.736,-179.483,8.805,149.564
C06470=1127.986,157.858,-60.755,-179.481,8.809,149.564
C06471=1127.982,158.073,-60.774,-179.479,8.812,149.564
C06472=1127.978,158.287,-60.793,-179.477,8.814,149.564
C06473=1127.974,158.502,-60.812,-179.475,8.817,149.564
C06474=1127.970,158.716,-60.831,-179.473,8.820,149.564
C06475=1127.966,158.965,-60.853,-179.470,8.824,149.564
C06476=1127.960,159.214,-60.876,-179.467,8.827,149.564
C06477=1127.956,159.463,-60.898,-179.465,8.830,149.565
C06478=1127.952,159.712,-60.920,-179.462,8.833,149.565
C06479=1127.947,159.961,-60.942,-179.460,8.836,149.565
C06480=1127.942,160.209,-60.965,-179.457,8.841,149.565
C06481=1127.938,160.459,-60.987,-179.455,8.844,149.565
C06482=1127.933,160.708,-61.009,-179.452,8.847,149.565
C06483=1127.928,160.957,-61.031,-179.450,8.850,149.565
C06484=1127.924,161.206,-61.054,-179.447,8.854,149.565
C06485=1127.919,161.454,-61.076,-179.445,8.857,149.565
C06486=1127.914,161.704,-61.098,-179.443,8.860,149.565
C06487=1127.910,161.953,-61.121,-179.440,8.864,149.565
C06488=1127.905,162.201,-61.143,-179.437,8.867,149.565
C06489=1127.900,162.450,-61.166,-179.435,8.870,149.566
C06490=1127.896,162.700,-61.188,-179.433,8.874,149.566
C06491=1127.891,162.948,-61.210,-179.430,8.877,149.566
C06492=1127.887,163.197,-61.233,-179.428,8.880,149.566
C06493=1127.882,163.447,-61.255,-179.425,8.883,149.566
C06494=1127.878,163.695,-61.278,-179.423,8.887,149.566
C06495=1127.873,163.944,-61.300,-179.420,8.890,149.566
C06496=1127.869,164.193,-61.323,-179.418,8.893,149.566
C06497=1127.863,164.442,-61.345,-179.416,8.896,149.566
C06498=1127.859,164.691,-61.368,-179.413,8.899,149.566
C06499=1127.854,164.941,-61.391,-179.411,8.902,149.566
C06500=1127.850,165.189,-61.413,-179.408,8.906,149.566
C06501=1127.845,165.438,-61.435,-179.406,8.909,149.567
C06502=1127.841,165.687,-61.459,-179.404,8.912,149.567
C06503=1127.836,165.935,-61.481,-179.401,8.915,149.567
C06504=1127.831,166.185,-61.504,-179.399,8.918,149.567
C06505=1127.827,166.433,-61.527,-179.396,8.922,149.567
C06506=1127.822,166.683,-61.549,-179.394,8.925,149.567
C06507=1127.818,166.931,-61.572,-179.391,8.928,149.567
C06508=1127.813,167.180,-61.595,-179.389,8.931,149.567
C06509=1127.808,167.430,-61.618,-179.387,8.935,149.567
C06510=1127.804,167.678,-61.640,-179.384,8.938,149.567
C06511=1127.799,167.927,-61.663,-179.382,8.940,149.567
C06512=1127.794,168.176,-61.685,-179.380,8.943,149.567
C06513=1127.790,168.425,-61.709,-179.378,8.947,149.568
C06514=1127.786,168.674,-61.731,-179.375,8.950,149.568
C06515=1127.780,168.923,-61.754,-179.373,8.953,149.568
C06516=1127.775,169.172,-61.777,-179.370,8.956,149.568
C06517=1127.771,169.421,-61.800,-179.368,8.959,149.568
C06518=1127.767,169.670,-61.823,-179.366,8.962,149.568
C06519=1127.762,169.918,-61.846,-179.364,8.965,149.568
C06520=1127.757,170.167,-61.868,-179.362,8.968,149.568
C06521=1127.753,170.416,-61.892,-179.359,8.971,149.568
C06522=1127.749,170.665,-61.914,-179.357,8.975,149.568
C06523=1127.744,170.879,-61.934,-179.355,8.977,149.568
C06524=1127.741,171.094,-61.954,-179.353,8.979,149.569
C06525=1127.736,171.308,-61.973,-179.351,8.983,149.569
C06526=1127.733,171.523,-61.994,-179.349,8.985,149.569
C06527=1127.728,171.737,-62.013,-179.347,8.987,149.569
C06528=1127.725,171.951,-62.034,-179.345,8.990,149.569
C06529=1127.720,172.165,-62.053,-179.343,8.993,149.569
C06530=1127.717,172.379,-62.073,-179.341,8.996,149.569
C06531=1127.712,172.629,-62.095,-179.339,8.999,149.569
C06532=1127.707,172.878,-62.119,-179.337,9.001,149.569
C06533=1127.702,173.127,-62.142,-179.335,9.004,149.569
C06534=1127.698,173.375,-62.165,-179.332,9.008,149.569
C06535=1127.694,173.625,-62.188,-179.329,9.011,149.569
C06536=1127.689,173.874,-62.212,-179.328,9.013,149.569
C06537=1127.684,174.123,-62.235,-179.325,9.016,149.570
C06538=1127.680,174.371,-62.257,-179.323,9.020,149.570
C06539=1127.675,174.620,-62.281,-179.321,9.022,149.570
C06540=1127.670,174.869,-62.304,-179.319,9.025,149.570
C06541=1127.666,175.118,-62.328,-179.316,9.029,149.570
C06542=1127.662,175.366,-62.350,-179.314,9.032,149.570
C06543=1127.657,175.615,-62.374,-179.312,9.034,149.570
C06544=1127.652,175.864,-62.397,-179.310,9.037,149.570
C06545=1127.648,176.114,-62.420,-179.307,9.041,149.570
C06546=1127.643,176.362,-62.444,-179.306,9.043,149.571
C06547=1127.639,176.611,-62.467,-179.303,9.046,149.571
C06548=1127.634,176.860,-62.491,-179.302,9.049,149.571
C06549=1127.630,177.109,-62.514,-179.299,9.052,149.571
C06550=1127.625,177.358,-62.537,-179.297,9.055,149.571
C06551=1127.620,177.606,-62.560,-179.295,9.058,149.571
C06552=1127.615,177.855,-62.584,-179.293,9.061,149.571
C06553=1127.610,178.104,-62.607,-179.290,9.064,149.571
C06554=1127.607,178.352,-62.630,-179.289,9.067,149.571
C06555=1127.602,178.601,-62.654,-179.286,9.070,149.572
C06556=1127.597,178.850,-62.677,-179.285,9.072,149.572
C06557=1127.593,179.099,-62.701,-179.282,9.075,149.572
C06558=1127.588,179.348,-62.725,-179.279,9.079,149.572
C06559=1127.583,179.597,-62.748,-179.276,9.082,149.572
C06560=1127.579,179.846,-62.771,-179.274,9.086,149.572
C06561=1127.574,180.095,-62.795,-179.270,9.089,149.572
C06562=1127.570,180.343,-62.819,-179.268,9.092,149.572
C06563=1127.565,180.592,-62.842,-179.265,9.096,149.572
C06564=1127.560,180.841,-62.865,-179.262,9.099,149.572
C06565=1127.556,181.090,-62.890,-179.258,9.103,149.572
C06566=1127.551,181.339,-62.913,-179.256,9.106,149.572
C06567=1127.547,181.588,-62.936,-179.253,9.109,149.572
C06568=1127.543,181.837,-62.961,-179.250,9.112,149.572
C06569=1127.538,182.086,-62.984,-179.247,9.115,149.572
C06570=1127.533,182.335,-63.007,-179.245,9.119,149.572
C06571=1127.529,182.583,-63.032,-179.242,9.122,149.572
C06572=1127.524,182.832,-63.055,-179.239,9.125,149.572
C06573=1127.520,183.081,-63.079,-179.236,9.128,149.572
C06574=1127.515,183.330,-63.102,-179.234,9.131,149.572
C06575=1127.511,183.578,-63.126,-179.231,9.134,149.571
C06576=1127.506,183.827,-63.150,-179.228,9.137,149.571
C06577=1127.502,184.076,-63.174,-179.226,9.140,149.572
C06578=1127.497,184.325,-63.197,-179.223,9.143,149.572
C06579=1127.493,184.539,-63.218,-179.221,9.147,149.572
C06580=1127.489,184.754,-63.239,-179.218,9.149,149.571
C06581=1127.485,184.967,-63.259,-179.216,9.152,149.571
C06582=1127.481,185.182,-63.279,-179.214,9.154,149.572
C06583=1127.478,185.397,-63.300,-179.211,9.157,149.572
C06584=1127.473,185.610,-63.321,-179.209,9.159,149.572
C06585=1127.469,185.824,-63.342,-179.207,9.162,149.572
C06586=1127.466,186.039,-63.362,-179.205,9.165,149.572
C06587=1127.462,186.288,-63.385,-179.203,9.167,149.571
C06588=1127.456,186.537,-63.410,-179.200,9.170,149.572
C06589=1127.452,186.785,-63.434,-179.198,9.173,149.572
C06590=1127.447,187.034,-63.458,-179.195,9.176,149.572
C06591=1127.443,187.283,-63.482,-179.193,9.178,149.572
C06592=1127.439,187.531,-63.506,-179.191,9.182,149.572
C06593=1127.434,187.781,-63.530,-179.188,9.185,149.572
C06594=1127.429,188.029,-63.554,-179.186,9.187,149.572
C06595=1127.425,188.278,-63.578,-179.184,9.190,149.572
C06596=1127.420,188.527,-63.602,-179.181,9.193,149.572
C06597=1127.416,188.776,-63.627,-179.179,9.196,149.572
C06598=1127.411,189.025,-63.651,-179.177,9.199,149.572
C06599=1127.407,189.273,-63.675,-179.175,9.201,149.572
C06600=1127.401,189.522,-63.699,-179.172,9.204,149.572
C06601=1127.397,189.771,-63.723,-179.170,9.206,149.572
C06602=1127.393,190.020,-63.747,-179.168,9.210,149.572
C06603=1127.389,190.268,-63.771,-179.166,9.212,149.572
C06604=1127.384,190.517,-63.796,-179.163,9.215,149.572
C06605=1127.379,190.766,-63.819,-179.162,9.218,149.572
C06606=1127.375,191.015,-63.844,-179.160,9.220,149.572
C06607=1127.370,191.264,-63.868,-179.158,9.223,149.573
C06608=1127.366,191.512,-63.892,-179.156,9.225,149.573
C06609=1127.361,191.761,-63.917,-179.154,9.228,149.573
C06610=1127.357,192.010,-63.942,-179.152,9.231,149.573
C06611=1127.352,192.258,-63.966,-179.150,9.234,149.573
C06612=1127.348,192.507,-63.990,-179.148,9.236,149.573
C06613=1127.343,192.756,-64.014,-179.146,9.239,149.573
C06614=1127.339,193.005,-64.038,-179.145,9.241,149.573
C06615=1127.334,193.254,-64.063,-179.142,9.244,149.573
C06616=1127.329,193.502,-64.087,-179.141,9.247,149.573
C06617=1127.325,193.752,-64.111,-179.139,9.249,149.573
C06618=1127.320,194.000,-64.136,-179.137,9.252,149.574
C06619=1127.316,194.249,-64.160,-179.135,9.254,149.574
C06620=1127.311,194.497,-64.185,-179.134,9.257,149.574
C06621=1127.307,194.747,-64.209,-179.132,9.259,149.574
C06622=1127.303,194.995,-64.233,-179.130,9.262,149.574
C06623=1127.297,195.244,-64.258,-179.129,9.265,149.575
C06624=1127.294,195.493,-64.282,-179.127,9.267,149.575
C06625=1127.289,195.742,-64.307,-179.126,9.270,149.575
C06626=1127.284,195.990,-64.331,-179.124,9.272,149.575
C06627=1127.280,196.239,-64.356,-179.122,9.275,149.575
C06628=1127.275,196.488,-64.380,-179.119,9.279,149.575
C06629=1127.271,196.736,-64.404,-179.116,9.282,149.575
C06630=1127.266,196.986,-64.429,-179.111,9.286,149.575
C06631=1127.262,197.233,-64.454,-179.108,9.290,149.575
C06632=1127.257,197.482,-64.479,-179.104,9.293,149.575
C06633=1127.253,197.731,-64.503,-179.101,9.297,149.574
C06634=1127.248,197.980,-64.528,-179.097,9.300,149.574
C06635=1127.245,198.194,-64.549,-179.093,9.304,149.574
C06636=1127.241,198.409,-64.570,-179.090,9.307,149.574
C06637=1127.237,198.622,-64.592,-179.087,9.310,149.574
C06638=1127.233,198.837,-64.614,-179.084,9.313,149.574
C06639=1127.229,199.051,-64.634,-179.081,9.316,149.574
C06640=1127.225,199.265,-64.656,-179.078,9.319,149.574
C06641=1127.221,199.479,-64.677,-179.075,9.322,149.573
C06642=1127.217,199.693,-64.698,-179.072,9.325,149.573
C06643=1127.213,199.942,-64.724,-179.068,9.329,149.573
C06644=1127.208,200.190,-64.748,-179.065,9.332,149.573
C06645=1127.204,200.440,-64.773,-179.062,9.335,149.573
C06646=1127.199,200.688,-64.798,-179.058,9.338,149.573
C06647=1127.195,200.936,-64.822,-179.055,9.342,149.573
C06648=1127.190,201.186,-64.847,-179.052,9.345,149.572
C06649=1127.185,201.434,-64.873,-179.048,9.348,149.572
C06650=1127.181,201.683,-64.897,-179.045,9.351,149.572
C06651=1127.177,201.931,-64.922,-179.042,9.354,149.572
C06652=1127.172,202.180,-64.947,-179.039,9.357,149.572
C06653=1127.168,202.428,-64.972,-179.035,9.361,149.572
C06654=1127.164,202.678,-64.997,-179.032,9.364,149.572
C06655=1127.159,202.926,-65.023,-179.029,9.367,149.572
C06656=1127.154,203.175,-65.048,-179.026,9.370,149.572
C06657=1127.151,203.424,-65.073,-179.023,9.373,149.571
C06658=1127.146,203.672,-65.097,-179.019,9.376,149.571
C06659=1127.141,203.921,-65.123,-179.016,9.379,149.571
C06660=1127.136,204.170,-65.148,-179.013,9.382,149.571
C06661=1127.132,204.419,-65.174,-179.011,9.385,149.571
C06662=1127.128,204.667,-65.198,-179.008,9.388,149.571
C06663=1127.123,204.916,-65.223,-179.005,9.390,149.571
C06664=1127.119,205.164,-65.249,-179.002,9.393,149.571
C06665=1127.114,205.414,-65.274,-179.000,9.396,149.571
C06666=1127.109,205.662,-65.299,-178.997,9.399,149.570
C06667=1127.105,205.911,-65.324,-178.994,9.402,149.570
C06668=1127.101,206.160,-65.349,-178.991,9.405,149.570
C06669=1127.096,206.408,-65.375,-178.988,9.407,149.570
C06670=1127.092,206.656,-65.401,-178.985,9.410,149.570
C06671=1127.087,206.905,-65.425,-178.983,9.413,149.570
C06672=1127.083,207.154,-65.451,-178.980,9.416,149.570
C06673=1127.078,207.403,-65.477,-178.978,9.418,149.570
C06674=1127.073,207.652,-65.501,-178.975,9.421,149.570
C06675=1127.069,207.900,-65.527,-178.972,9.424,149.570
C06676=1127.064,208.148,-65.553,-178.969,9.427,149.570
C06677=1127.060,208.397,-65.578,-178.968,9.429,149.570
C06678=1127.056,208.646,-65.604,-178.965,9.432,149.570
C06679=1127.051,208.895,-65.629,-178.963,9.434,149.570
C06680=1127.047,209.144,-65.654,-178.960,9.437,149.570
C06681=1127.043,209.392,-65.680,-178.958,9.440,149.570
C06682=1127.038,209.640,-65.705,-178.956,9.443,149.570
C06683=1127.034,209.889,-65.731,-178.954,9.445,149.570
C06684=1127.030,210.138,-65.757,-178.951,9.448,149.570
C06685=1127.025,210.386,-65.781,-178.949,9.451,149.570
C06686=1127.020,210.635,-65.807,-178.947,9.454,149.570
C06687=1127.016,210.884,-65.833,-178.945,9.456,149.570
C06688=1127.011,211.132,-65.858,-178.943,9.458,149.570
C06689=1127.006,211.381,-65.884,-178.941,9.462,149.570
C06690=1127.002,211.630,-65.910,-178.939,9.464,149.570
C06691=1126.999,211.844,-65.932,-178.937,9.466,149.570
C06692=1126.994,212.058,-65.954,-178.935,9.469,149.570
C06693=1126.991,212.272,-65.976,-178.934,9.470,149.571
C06694=1126.987,212.486,-65.998,-178.932,9.473,149.571
C06695=1126.983,212.699,-66.020,-178.930,9.475,149.571
C06696=1126.979,212.914,-66.042,-178.929,9.477,149.571
C06697=1126.976,213.128,-66.064,-178.928,9.479,149.571
C06698=1126.972,213.342,-66.087,-178.926,9.482,149.571
C06699=1126.967,213.590,-66.112,-178.924,9.484,149.571
C06700=1126.963,213.839,-66.138,-178.923,9.487,149.572
C06701=1126.959,214.088,-66.164,-178.921,9.489,149.572
C06702=1126.954,214.336,-66.190,-178.918,9.493,149.572
C06703=1126.950,214.584,-66.215,-178.917,9.495,149.572
C06704=1126.945,214.833,-66.241,-178.915,9.498,149.572
C06705=1126.940,215.082,-66.267,-178.913,9.501,149.572
C06706=1126.936,215.331,-66.293,-178.911,9.503,149.572
C06707=1126.931,215.579,-66.318,-178.909,9.507,149.572
C06708=1126.927,215.828,-66.344,-178.907,9.509,149.573
C06709=1126.923,216.077,-66.370,-178.904,9.512,149.573
C06710=1126.919,216.326,-66.395,-178.903,9.515,149.573
C06711=1126.915,216.574,-66.422,-178.900,9.518,149.573
C06712=1126.909,216.822,-66.448,-178.899,9.520,149.573
C06713=1126.905,217.071,-66.474,-178.896,9.524,149.573
C06714=1126.901,217.320,-66.499,-178.894,9.527,149.573
C06715=1126.896,217.569,-66.525,-178.892,9.529,149.573
C06716=1126.893,217.817,-66.552,-178.890,9.533,149.574
C06717=1126.887,218.065,-66.578,-178.887,9.536,149.574
C06718=1126.883,218.314,-66.603,-178.885,9.539,149.574
C06719=1126.879,218.563,-66.629,-178.883,9.541,149.574
C06720=1126.874,218.812,-66.655,-178.881,9.545,149.574
C06721=1126.870,219.060,-66.682,-178.878,9.548,149.574
C06722=1126.865,219.309,-66.708,-178.876,9.551,149.574
C06723=1126.861,219.557,-66.733,-178.873,9.554,149.574
C06724=1126.857,219.805,-66.759,-178.871,9.557,149.574
C06725=1126.852,220.054,-66.786,-178.868,9.560,149.574
C06726=1126.847,220.303,-66.812,-178.866,9.563,149.574
C06727=1126.844,220.551,-66.838,-178.864,9.567,149.575
C06728=1126.839,220.800,-66.864,-178.861,9.570,149.575
C06729=1126.834,221.049,-66.890,-178.859,9.573,149.575
C06730=1126.830,221.297,-66.916,-178.856,9.576,149.575
C06731=1126.826,221.546,-66.942,-178.853,9.579,149.575
C06732=1126.821,221.795,-66.968,-178.851,9.582,149.575
C06733=1126.817,222.043,-66.995,-178.848,9.585,149.575
C06734=1126.812,222.292,-67.021,-178.845,9.589,149.575
C06735=1126.808,222.540,-67.048,-178.842,9.592,149.575
C06736=1126.804,222.789,-67.073,-178.840,9.595,149.575
C06737=1126.799,223.038,-67.100,-178.837,9.598,149.575
C06738=1126.795,223.286,-67.126,-178.834,9.602,149.575
C06739=1126.790,223.535,-67.153,-178.831,9.605,149.575
C06740=1126.785,223.783,-67.179,-178.829,9.608,149.575
C06741=1126.781,224.031,-67.205,-178.825,9.612,149.575
C06742=1126.776,224.280,-67.231,-178.822,9.615,149.575
C06743=1126.772,224.528,-67.258,-178.819,9.619,149.575
C06744=1126.768,224.778,-67.284,-178.817,9.622,149.575
C06745=1126.764,225.026,-67.311,-178.813,9.625,149.575
C06746=1126.759,225.274,-67.338,-178.811,9.628,149.575
C06747=1126.755,225.489,-67.360,-178.808,9.631,149.575
C06748=1126.752,225.703,-67.382,-178.805,9.634,149.575
C06749=1126.748,225.916,-67.405,-178.802,9.637,149.575
C06750=1126.744,226.130,-67.428,-178.800,9.640,149.575
C06751=1126.740,226.344,-67.451,-178.797,9.643,149.575
C06752=1126.736,226.558,-67.474,-178.794,9.646,149.575
C06753=1126.732,226.772,-67.497,-178.791,9.649,149.575
C06754=1126.729,226.986,-67.520,-178.789,9.652,149.575
C06755=1126.724,227.234,-67.547,-178.786,9.655,149.575
C06756=1126.720,227.483,-67.573,-178.782,9.658,149.575
C06757=1126.715,227.732,-67.600,-178.779,9.662,149.574
C06758=1126.711,227.980,-67.626,-178.775,9.665,149.574
C06759=1126.707,228.228,-67.653,-178.773,9.668,149.574
C06760=1126.703,228.477,-67.680,-178.769,9.672,149.574
C06761=1126.698,228.725,-67.707,-178.765,9.675,149.574
C06762=1126.693,228.974,-67.733,-178.762,9.679,149.574
C06763=1126.689,229.222,-67.760,-178.758,9.682,149.574
C06764=1126.685,229.471,-67.787,-178.755,9.686,149.574
C06765=1126.680,229.719,-67.814,-178.751,9.689,149.574
C06766=1126.677,229.968,-67.841,-178.747,9.693,149.573
C06767=1126.672,230.217,-67.868,-178.744,9.695,149.573
C06768=1126.667,230.465,-67.895,-178.741,9.699,149.573
C06769=1126.663,230.713,-67.921,-178.737,9.702,149.573
C06770=1126.659,230.962,-67.948,-178.733,9.706,149.573
C06771=1126.654,231.210,-67.975,-178.729,9.709,149.573
C06772=1126.649,231.459,-68.002,-178.726,9.712,149.573
C06773=1126.646,231.707,-68.029,-178.723,9.715,149.572
C06774=1126.641,231.956,-68.056,-178.720,9.718,149.572
C06775=1126.637,232.205,-68.083,-178.716,9.722,149.572
C06776=1126.632,232.453,-68.110,-178.713,9.724,149.572
C06777=1126.628,232.701,-68.137,-178.710,9.728,149.572
C06778=1126.624,232.950,-68.164,-178.707,9.731,149.572
C06779=1126.619,233.198,-68.191,-178.704,9.733,149.572
C06780=1126.615,233.448,-68.218,-178.700,9.737,149.572
C06781=1126.611,233.695,-68.246,-178.697,9.739,149.571
C06782=1126.607,233.944,-68.273,-178.694,9.742,149.571
C06783=1126.602,234.192,-68.300,-178.691,9.745,149.571
C06784=1126.597,234.441,-68.327,-178.687,9.748,149.571
C06785=1126.593,234.690,-68.354,-178.685,9.751,149.571
C06786=1126.589,234.938,-68.382,-178.682,9.754,149.571
C06787=1126.584,235.186,-68.409,-178.679,9.756,149.571
C06788=1126.580,235.435,-68.436,-178.676,9.759,149.570
C06789=1126.575,235.683,-68.463,-178.673,9.762,149.570
C06790=1126.572,235.931,-68.491,-178.670,9.765,149.570
C06791=1126.567,236.180,-68.518,-178.667,9.768,149.570
C06792=1126.563,236.428,-68.545,-178.664,9.771,149.570
C06793=1126.558,236.677,-68.572,-178.662,9.773,149.570
C06794=1126.554,236.926,-68.600,-178.659,9.775,149.570
C06795=1126.550,237.174,-68.627,-178.656,9.778,149.570
C06796=1126.545,237.423,-68.654,-178.653,9.781,149.570
C06797=1126.541,237.671,-68.682,-178.651,9.783,149.570
C06798=1126.536,237.920,-68.709,-178.648,9.786,149.569
C06799=1126.532,238.167,-68.737,-178.645,9.789,149.569
C06800=1126.527,238.416,-68.764,-178.643,9.791,149.569
C06801=1126.523,238.665,-68.792,-178.641,9.794,149.569
C06802=1126.519,238.913,-68.819,-178.638,9.796,149.569
C06803=1126.516,239.127,-68.843,-178.636,9.798,149.569
C06804=1126.511,239.341,-68.867,-178.634,9.800,149.569
C06805=1126.508,239.554,-68.890,-178.632,9.802,149.569
C06806=1126.504,239.768,-68.913,-178.630,9.804,149.569
C06807=1126.500,239.982,-68.938,-178.627,9.806,149.569
C06808=1126.497,240.196,-68.962,-178.626,9.809,149.569
C06809=1126.493,240.410,-68.984,-178.624,9.811,149.569
C06810=1126.489,240.624,-69.009,-178.621,9.813,149.569
C06811=1126.485,240.871,-69.037,-178.619,9.815,149.569
C06812=1126.480,241.120,-69.064,-178.617,9.817,149.569
C06813=1126.476,241.369,-69.092,-178.615,9.820,149.569
C06814=1126.472,241.617,-69.119,-178.613,9.823,149.569
C06815=1126.467,241.865,-69.147,-178.610,9.825,149.569
C06816=1126.463,242.114,-69.174,-178.609,9.827,149.569
C06817=1126.459,242.362,-69.202,-178.607,9.829,149.569
C06818=1126.454,242.611,-69.231,-178.605,9.832,149.569
C06819=1126.450,242.859,-69.258,-178.602,9.834,149.569
C06820=1126.445,243.107,-69.285,-178.601,9.836,149.569
C06821=1126.441,243.356,-69.313,-178.599,9.838,149.569
C06822=1126.437,243.604,-69.341,-178.597,9.841,149.569
C06823=1126.433,243.852,-69.368,-178.595,9.843,149.569
C06824=1126.429,244.101,-69.396,-178.593,9.845,149.569
C06825=1126.423,244.350,-69.424,-178.591,9.848,149.569
C06826=1126.420,244.598,-69.452,-178.589,9.850,149.569
C06827=1126.415,244.847,-69.479,-178.588,9.852,149.569
C06828=1126.411,245.095,-69.507,-178.586,9.854,149.569
C06829=1126.407,245.343,-69.535,-178.585,9.857,149.570
C06830=1126.403,245.591,-69.563,-178.583,9.859,149.570
C06831=1126.398,245.841,-69.591,-178.582,9.861,149.570
C06832=1126.393,246.088,-69.619,-178.580,9.863,149.570
C06833=1126.390,246.337,-69.647,-178.578,9.865,149.570
C06834=1126.385,246.585,-69.674,-178.577,9.867,149.570
C06835=1126.381,246.833,-69.702,-178.575,9.870,149.570
C06836=1126.376,247.082,-69.731,-178.574,9.872,149.570
C06837=1126.372,247.330,-69.758,-178.573,9.874,149.571
C06838=1126.368,247.579,-69.786,-178.568,9.878,149.570
C06839=1126.363,247.827,-69.814,-178.562,9.883,149.570
C06840=1126.359,248.076,-69.842,-178.556,9.889,149.570
C06841=1126.355,248.324,-69.870,-178.549,9.893,149.569
C06842=1126.351,248.572,-69.898,-178.543,9.898,149.568
C06843=1126.346,248.821,-69.927,-178.538,9.902,149.568
C06844=1126.342,249.069,-69.955,-178.532,9.906,149.568
C06845=1126.338,249.317,-69.983,-178.527,9.911,149.567
C06846=1126.333,249.566,-70.011,-178.522,9.915,149.567
C06847=1126.329,249.814,-70.039,-178.516,9.919,149.566
C06848=1126.325,250.062,-70.067,-178.511,9.923,149.566
C06849=1126.320,250.311,-70.096,-178.507,9.926,149.566
C06850=1126.316,250.559,-70.124,-178.502,9.930,149.565
C06851=1126.311,250.807,-70.152,-178.498,9.933,149.565
C06852=1126.307,251.056,-70.180,-178.494,9.936,149.565
C06853=1126.303,251.305,-70.209,-178.491,9.939,149.564
C06854=1126.299,251.553,-70.237,-178.487,9.942,149.564
C06855=1126.294,251.802,-70.266,-178.484,9.944,149.564
C06856=1126.290,252.049,-70.294,-178.481,9.947,149.564
C06857=1126.286,252.298,-70.323,-178.478,9.950,149.564
C06858=1126.282,252.546,-70.351,-178.475,9.952,149.564
C06859=1126.277,252.760,-70.375,-178.473,9.954,149.563
C06860=1126.274,252.973,-70.400,-178.471,9.956,149.563
C06861=1126.271,253.187,-70.424,-178.470,9.957,149.563
C06862=1126.267,253.401,-70.449,-178.468,9.959,149.563
C06863=1126.263,253.614,-70.474,-178.466,9.961,149.563
C06864=1126.259,253.828,-70.498,-178.465,9.962,149.563
C06865=1126.256,254.041,-70.522,-178.463,9.964,149.563
C06866=1126.252,254.255,-70.547,-178.463,9.964,149.563
C06867=1126.248,254.504,-70.576,-178.462,9.966,149.563
C06868=1126.244,254.752,-70.604,-178.461,9.967,149.564
C06869=1126.239,255.000,-70.633,-178.460,9.969,149.564
C06870=1126.235,255.248,-70.661,-178.460,9.970,149.564
C06871=1126.230,255.497,-70.689,-178.461,9.971,149.564
C06872=1126.226,255.745,-70.717,-178.460,9.972,149.564
C06873=1126.222,255.993,-70.747,-178.460,9.973,149.565
C06874=1126.217,256.242,-70.775,-178.458,9.976,149.565
C06875=1126.213,256.490,-70.803,-178.455,9.979,149.565
C06876=1126.209,256.738,-70.833,-178.452,9.981,149.565
C06877=1126.205,256.986,-70.861,-178.449,9.984,149.564
C06878=1126.200,257.235,-70.889,-178.446,9.987,149.564
C06879=1126.196,257.484,-70.919,-178.443,9.990,149.564
C06880=1126.192,257.731,-70.947,-178.440,9.993,149.564
C06881=1126.187,257.980,-70.975,-178.438,9.996,149.564
C06882=1126.184,258.228,-71.004,-178.434,9.999,149.564
C06883=1126.179,258.476,-71.033,-178.431,10.002,149.564
C06884=1126.175,258.725,-71.062,-178.428,10.005,149.564
C06885=1126.171,258.973,-71.090,-178.425,10.007,149.564
C06886=1126.167,259.222,-71.120,-178.422,10.011,149.564
C06887=1126.162,259.470,-71.148,-178.418,10.013,149.563
C06888=1126.158,259.718,-71.177,-178.415,10.016,149.563
C06889=1126.154,259.967,-71.206,-178.412,10.020,149.563
C06890=1126.150,260.215,-71.235,-178.409,10.022,149.563
C06891=1126.144,260.463,-71.263,-178.406,10.025,149.563
C06892=1126.141,260.711,-71.292,-178.402,10.029,149.563
C06893=1126.137,260.960,-71.321,-178.399,10.031,149.563
C06894=1126.132,261.208,-71.351,-178.395,10.035,149.562
C06895=1126.128,261.456,-71.380,-178.392,10.037,149.562
C06896=1126.124,261.704,-71.408,-178.388,10.041,149.562
C06897=1126.120,261.953,-71.437,-178.385,10.043,149.562
C06898=1126.115,262.201,-71.466,-178.381,10.046,149.562
C06899=1126.111,262.450,-71.495,-178.379,10.049,149.562
C06900=1126.106,262.697,-71.524,-178.375,10.052,149.561
C06901=1126.102,262.946,-71.553,-178.371,10.056,149.561
C06902=1126.098,263.194,-71.582,-178.368,10.058,149.561
C06903=1126.094,263.442,-71.612,-178.364,10.062,149.561
C06904=1126.090,263.691,-71.641,-178.360,10.065,149.561
C06905=1126.085,263.939,-71.669,-178.357,10.067,149.560
C06906=1126.081,264.187,-71.699,-178.353,10.071,149.560
C06907=1126.076,264.435,-71.728,-178.349,10.074,149.560
C06908=1126.072,264.684,-71.758,-178.346,10.077,149.560
C06909=1126.068,264.932,-71.787,-178.344,10.079,149.560
C06910=1126.064,265.180,-71.815,-178.342,10.081,149.560
C06911=1126.060,265.428,-71.844,-178.339,10.084,149.559
C06912=1126.055,265.676,-71.874,-178.336,10.086,149.559
C06913=1126.051,265.925,-71.903,-178.333,10.088,149.559
C06914=1126.047,266.173,-71.933,-178.331,10.090,149.559
C06915=1126.043,266.386,-71.958,-178.329,10.092,149.559
C06916=1126.040,266.600,-71.983,-178.327,10.095,149.559
C06917=1126.036,266.813,-72.009,-178.325,10.097,149.559
C06918=1126.032,267.027,-72.034,-178.322,10.099,149.559
C06919=1126.028,267.240,-72.059,-178.320,10.101,149.559
C06920=1126.025,267.454,-72.084,-178.318,10.103,149.558
C06921=1126.021,267.667,-72.110,-178.316,10.105,149.559
C06922=1126.018,267.881,-72.135,-178.313,10.108,149.558
C06923=1126.014,268.129,-72.164,-178.311,10.110,149.558
C06924=1126.009,268.377,-72.194,-178.308,10.112,149.558
C06925=1126.005,268.625,-72.223,-178.305,10.114,149.558
C06926=1126.001,268.874,-72.253,-178.302,10.117,149.558
C06927=1125.997,269.122,-72.282,-178.299,10.120,149.558
C06928=1125.993,269.370,-72.312,-178.297,10.122,149.558
C06929=1125.988,269.619,-72.342,-178.294,10.125,149.558
C06930=1125.984,269.867,-72.371,-178.291,10.127,149.558
C06931=1125.979,270.115,-72.400,-178.288,10.130,149.557
C06932=1125.975,270.364,-72.430,-178.286,10.132,149.557
C06933=1125.971,270.612,-72.459,-178.283,10.135,149.557
C06934=1125.967,270.860,-72.489,-178.280,10.138,149.557
C06935=1125.963,271.108,-72.518,-178.277,10.140,149.557
C06936=1125.959,271.356,-72.548,-178.274,10.143,149.557
C06937=1125.955,271.604,-72.578,-178.272,10.145,149.557
C06938=1125.950,271.852,-72.607,-178.269,10.148,149.557
C06939=1125.945,272.101,-72.637,-178.266,10.151,149.557
C06940=1125.941,272.349,-72.667,-178.263,10.153,149.557
C06941=1125.937,272.598,-72.696,-178.260,10.156,149.556
C06942=1125.933,272.845,-72.727,-178.257,10.159,149.556
C06943=1125.929,273.094,-72.756,-178.254,10.162,149.556
C06944=1125.925,273.342,-72.785,-178.251,10.164,149.556
C06945=1125.920,273.590,-72.815,-178.248,10.167,149.556
C06946=1125.916,273.838,-72.846,-178.245,10.170,149.556
C06947=1125.912,274.086,-72.875,-178.242,10.172,149.556
C06948=1125.908,274.335,-72.905,-178.239,10.175,149.556
C06949=1125.904,274.582,-72.935,-178.236,10.178,149.555
C06950=1125.899,274.831,-72.965,-178.233,10.180,149.555
C06951=1125.895,275.079,-72.994,-178.230,10.183,149.555
C06952=1125.891,275.327,-73.024,-178.227,10.186,149.555
C06953=1125.887,275.575,-73.054,-178.224,10.189,149.555
C06954=1125.882,275.823,-73.085,-178.221,10.191,149.555
C06955=1125.878,276.072,-73.114,-178.218,10.194,149.554
C06956=1125.874,276.320,-73.144,-178.215,10.197,149.554
C06957=1125.870,276.568,-73.175,-178.211,10.199,149.554
C06958=1125.865,276.816,-73.204,-178.209,10.202,149.554
C06959=1125.862,277.064,-73.234,-178.205,10.205,149.554
C06960=1125.857,277.312,-73.264,-178.202,10.208,149.554
C06961=1125.853,277.560,-73.294,-178.199,10.210,149.554
C06962=1125.849,277.809,-73.324,-178.195,10.213,149.553
C06963=1125.845,278.057,-73.354,-178.192,10.216,149.553
C06964=1125.840,278.305,-73.385,-178.188,10.219,149.553
C06965=1125.837,278.553,-73.415,-178.186,10.222,149.553
C06966=1125.832,278.801,-73.445,-178.182,10.224,149.552
C06967=1125.828,279.049,-73.475,-178.179,10.227,149.552
C06968=1125.824,279.297,-73.505,-178.175,10.230,149.552
C06969=1125.820,279.546,-73.535,-178.172,10.233,149.552
C06970=1125.816,279.794,-73.566,-178.169,10.235,149.552
C06971=1125.812,280.007,-73.592,-178.166,10.238,149.552
C06972=1125.808,280.220,-73.617,-178.163,10.240,149.551
C06973=1125.804,280.434,-73.644,-178.160,10.242,149.551
C06974=1125.801,280.648,-73.669,-178.157,10.245,149.551
C06975=1125.797,280.861,-73.696,-178.154,10.247,149.551
C06976=1125.794,281.074,-73.722,-178.151,10.250,149.551
C06977=1125.790,281.288,-73.748,-178.148,10.252,149.550
C06978=1125.786,281.501,-73.774,-178.145,10.255,149.550
C06979=1125.782,281.749,-73.805,-178.142,10.257,149.550
C06980=1125.778,281.997,-73.835,-178.139,10.260,149.550
C06981=1125.774,282.245,-73.865,-178.136,10.263,149.550
C06982=1125.770,282.494,-73.896,-178.133,10.265,149.550
C06983=1125.766,282.741,-73.926,-178.130,10.268,149.549
C06984=1125.761,282.989,-73.957,-178.127,10.269,149.549
C06985=1125.757,283.237,-73.987,-178.124,10.272,149.549
C06986=1125.753,283.486,-74.018,-178.121,10.275,149.549
C06987=1125.749,283.734,-74.048,-178.118,10.277,149.549
C06988=1125.744,283.982,-74.078,-178.115,10.280,149.549
C06989=1125.740,284.230,-74.109,-178.112,10.282,149.548
C06990=1125.736,284.478,-74.140,-178.109,10.285,149.548
C06991=1125.732,284.726,-74.170,-178.106,10.288,149.548
C06992=1125.728,284.974,-74.201,-178.103,10.290,149.548
C06993=1125.724,285.222,-74.232,-178.099,10.293,149.548
C06994=1125.719,285.470,-74.262,-178.097,10.295,149.547
C06995=1125.716,285.718,-74.293,-178.094,10.298,149.547
C06996=1125.711,285.967,-74.324,-178.091,10.300,149.547
C06997=1125.707,286.215,-74.355,-178.088,10.303,149.547
C06998=1125.703,286.462,-74.385,-178.084,10.305,149.547
C06999=1125.699,286.711,-74.416,-178.081,10.308,149.547
C07000=1125.694,286.959,-74.447,-178.078,10.310,149.546
C07001=1125.691,287.206,-74.477,-178.075,10.313,149.546
C07002=1125.686,287.455,-74.508,-178.072,10.316,149.546
C07003=1125.682,287.703,-74.539,-178.069,10.318,149.546
C07004=1125.677,287.951,-74.569,-178.067,10.320,149.546
C07005=1125.674,288.199,-74.600,-178.063,10.323,149.546
C07006=1125.670,288.447,-74.631,-178.060,10.325,149.545
C07007=1125.665,288.695,-74.662,-178.057,10.328,149.545
C07008=1125.661,288.943,-74.693,-178.054,10.331,149.545
C07009=1125.657,289.191,-74.723,-178.051,10.333,149.545
C07010=1125.653,289.440,-74.755,-178.048,10.336,149.545
C07011=1125.649,289.688,-74.785,-178.044,10.338,149.544
C07012=1125.644,289.935,-74.817,-178.041,10.341,149.544
C07013=1125.641,290.183,-74.847,-178.039,10.344,149.544
C07014=1125.636,290.431,-74.878,-178.036,10.345,149.544
C07015=1125.632,290.680,-74.909,-178.033,10.348,149.544
C07016=1125.628,290.927,-74.941,-178.030,10.351,149.544
C07017=1125.624,291.176,-74.972,-178.027,10.353,149.543
C07018=1125.619,291.424,-75.003,-178.023,10.356,149.543
C07019=1125.616,291.671,-75.034,-178.020,10.359,149.543
C07020=1125.612,291.920,-75.065,-178.017,10.361,149.543
C07021=1125.607,292.168,-75.095,-178.014,10.364,149.543
C07022=1125.604,292.416,-75.127,-178.011,10.366,149.542
C07023=1125.599,292.664,-75.158,-178.008,10.369,149.542
C07024=1125.595,292.912,-75.189,-178.004,10.371,149.542
C07025=1125.591,293.160,-75.221,-178.002,10.373,149.542
C07026=1125.587,293.408,-75.252,-177.999,10.376,149.542
C07027=1125.584,293.620,-75.278,-177.996,10.379,149.542
C07028=1125.580,293.834,-75.305,-177.994,10.381,149.542
C07029=1125.576,294.047,-75.332,-177.991,10.383,149.541
C07030=1125.573,294.261,-75.359,-177.988,10.385,149.541
C07031=1125.569,294.474,-75.386,-177.986,10.387,149.541
C07032=1125.566,294.687,-75.413,-177.983,10.390,149.541
C07033=1125.562,294.900,-75.440,-177.980,10.392,149.541
C07034=1125.559,295.114,-75.467,-177.978,10.393,149.541
C07035=1125.554,295.362,-75.498,-177.975,10.396,149.540
C07036=1125.550,295.610,-75.529,-177.971,10.399,149.540
C07037=1125.546,295.857,-75.561,-177.969,10.401,149.540
C07038=1125.542,296.106,-75.592,-177.965,10.404,149.540
C07039=1125.538,296.353,-75.623,-177.962,10.407,149.540
C07040=1125.534,296.602,-75.655,-177.959,10.409,149.539
C07041=1125.529,296.849,-75.686,-177.956,10.412,149.539
C07042=1125.526,297.097,-75.718,-177.953,10.414,149.539
C07043=1125.522,297.346,-75.749,-177.950,10.417,149.539
C07044=1125.517,297.593,-75.781,-177.947,10.419,149.539
C07045=1125.513,297.842,-75.812,-177.944,10.421,149.539
C07046=1125.509,298.089,-75.843,-177.941,10.424,149.538
C07047=1125.505,298.337,-75.875,-177.938,10.426,149.538
C07048=1125.500,298.585,-75.907,-177.934,10.429,149.538
C07049=1125.496,298.833,-75.938,-177.932,10.432,149.538
C07050=1125.493,299.081,-75.970,-177.928,10.434,149.538
C07051=1125.488,299.329,-76.001,-177.925,10.437,149.538
C07052=1125.484,299.577,-76.033,-177.922,10.439,149.537
C07053=1125.481,299.825,-76.064,-177.919,10.442,149.537
C07054=1125.476,300.073,-76.096,-177.916,10.445,149.537
C07055=1125.473,300.321,-76.128,-177.913,10.447,149.537
C07056=1125.467,300.569,-76.160,-177.910,10.449,149.537
C07057=1125.463,300.817,-76.191,-177.907,10.452,149.537
C07058=1125.460,301.065,-76.223,-177.904,10.454,149.536
C07059=1125.455,301.313,-76.254,-177.901,10.457,149.536
C07060=1125.452,301.561,-76.286,-177.897,10.459,149.536
C07061=1125.447,301.809,-76.319,-177.895,10.462,149.536
C07062=1125.443,302.056,-76.350,-177.891,10.465,149.536
C07063=1125.439,302.304,-76.382,-177.888,10.467,149.535
C07064=1125.436,302.552,-76.414,-177.885,10.470,149.535
C07065=1125.431,302.800,-76.446,-177.882,10.472,149.535
C07066=1125.427,303.048,-76.478,-177.879,10.475,149.535
C07067=1125.423,303.296,-76.510,-177.876,10.478,149.535
C07068=1125.418,303.544,-76.541,-177.873,10.479,149.534
C07069=1125.414,303.792,-76.573,-177.870,10.482,149.534
C07070=1125.410,304.040,-76.605,-177.867,10.485,149.534
C07071=1125.406,304.287,-76.637,-177.863,10.487,149.534
C07072=1125.402,304.535,-76.669,-177.861,10.490,149.534
C07073=1125.398,304.784,-76.701,-177.857,10.492,149.534
C07074=1125.395,305.032,-76.733,-177.854,10.495,149.533
C07075=1125.389,305.279,-76.765,-177.851,10.497,149.533
C07076=1125.386,305.527,-76.797,-177.848,10.500,149.533
C07077=1125.381,305.776,-76.829,-177.845,10.503,149.533
C07078=1125.378,306.024,-76.861,-177.842,10.505,149.533
C07079=1125.373,306.271,-76.893,-177.838,10.508,149.533
C07080=1125.369,306.519,-76.925,-177.835,10.511,149.532
C07081=1125.365,306.767,-76.958,-177.833,10.512,149.532
C07082=1125.361,307.015,-76.990,-177.829,10.515,149.532
C07083=1125.357,307.228,-77.017,-177.827,10.517,149.532
C07084=1125.354,307.441,-77.045,-177.824,10.519,149.532
C07085=1125.351,307.654,-77.072,-177.821,10.522,149.531
C07086=1125.347,307.867,-77.100,-177.819,10.524,149.531
C07087=1125.344,308.080,-77.128,-177.816,10.526,149.531
C07088=1125.340,308.293,-77.156,-177.813,10.528,149.531
C07089=1125.336,308.506,-77.183,-177.811,10.530,149.531
C07090=1125.333,308.719,-77.211,-177.808,10.532,149.531
C07091=1125.329,308.967,-77.243,-177.805,10.535,149.531
C07092=1125.325,309.216,-77.275,-177.802,10.537,149.530
C07093=1125.321,309.463,-77.308,-177.799,10.540,149.530
C07094=1125.316,309.711,-77.340,-177.795,10.542,149.530
C07095=1125.312,309.959,-77.372,-177.793,10.545,149.530
C07096=1125.309,310.206,-77.405,-177.789,10.548,149.530
C07097=1125.304,310.455,-77.437,-177.786,10.550,149.530
C07098=1125.301,310.702,-77.470,-177.783,10.553,149.529
C07099=1125.296,310.950,-77.502,-177.780,10.556,149.529
C07100=1125.293,311.199,-77.534,-177.777,10.558,149.529
C07101=1125.288,311.446,-77.567,-177.773,10.560,149.529
C07102=1125.284,311.694,-77.599,-177.770,10.563,149.529
C07103=1125.280,311.941,-77.632,-177.768,10.565,149.528
C07104=1125.276,312.190,-77.664,-177.765,10.568,149.528
C07105=1125.272,312.437,-77.697,-177.761,10.570,149.528
C07106=1125.268,312.685,-77.729,-177.759,10.573,149.528
C07107=1125.264,312.933,-77.762,-177.755,10.575,149.528
C07108=1125.260,313.181,-77.794,-177.752,10.578,149.527
C07109=1125.256,313.429,-77.827,-177.749,10.580,149.527
C07110=1125.252,313.677,-77.859,-177.746,10.583,149.527
C07111=1125.247,313.924,-77.892,-177.743,10.586,149.527
C07112=1125.243,314.172,-77.925,-177.739,10.588,149.527
C07113=1125.239,314.420,-77.957,-177.736,10.591,149.526
C07114=1125.235,314.667,-77.990,-177.733,10.593,149.526
C07115=1125.231,314.916,-78.023,-177.730,10.596,149.526
C07116=1125.227,315.163,-78.055,-177.727,10.599,149.526
C07117=1125.223,315.411,-78.088,-177.724,10.600,149.526
C07118=1125.219,315.659,-78.121,-177.721,10.603,149.526
C07119=1125.215,315.907,-78.153,-177.718,10.605,149.525
C07120=1125.211,316.154,-78.186,-177.715,10.608,149.525
C07121=1125.207,316.402,-78.220,-177.712,10.611,149.525
C07122=1125.203,316.651,-78.252,-177.708,10.613,149.525
C07123=1125.199,316.898,-78.285,-177.705,10.615,149.525
C07124=1125.195,317.146,-78.318,-177.702,10.618,149.525
C07125=1125.191,317.393,-78.351,-177.699,10.621,149.524
C07126=1125.187,317.642,-78.383,-177.695,10.623,149.524
C07127=1125.183,317.889,-78.416,-177.692,10.626,149.524
C07128=1125.179,318.137,-78.449,-177.689,10.628,149.524
C07129=1125.175,318.385,-78.482,-177.686,10.631,149.524
C07130=1125.171,318.632,-78.515,-177.683,10.634,149.523
C07131=1125.167,318.880,-78.549,-177.680,10.636,149.523
C07132=1125.163,319.128,-78.580,-177.677,10.638,149.523
C07133=1125.159,319.376,-78.614,-177.674,10.640,149.523
C07134=1125.155,319.624,-78.647,-177.671,10.643,149.523
C07135=1125.151,319.871,-78.680,-177.668,10.646,149.522
C07136=1125.147,320.120,-78.713,-177.664,10.648,149.522
C07137=1125.143,320.368,-78.747,-177.661,10.651,149.522
C07138=1125.139,320.615,-78.779,-177.658,10.653,149.522
C07139=1125.136,320.828,-78.808,-177.655,10.655,149.522
C07140=1125.132,321.041,-78.836,-177.653,10.658,149.522
C07141=1125.128,321.254,-78.865,-177.650,10.660,149.521
C07142=1125.125,321.466,-78.893,-177.647,10.662,149.521
C07143=1125.122,321.679,-78.922,-177.645,10.664,149.521
C07144=1125.118,321.892,-78.950,-177.642,10.666,149.521
C07145=1125.115,322.105,-78.978,-177.639,10.669,149.521
C07146=1125.112,322.318,-79.007,-177.636,10.670,149.521
C07147=1125.107,322.566,-79.040,-177.633,10.673,149.520
C07148=1125.103,322.813,-79.073,-177.630,10.676,149.520
C07149=1125.100,323.062,-79.107,-177.627,10.678,149.520
C07150=1125.096,323.310,-79.140,-177.624,10.681,149.520
C07151=1125.091,323.557,-79.173,-177.620,10.683,149.520
C07152=1125.087,323.805,-79.206,-177.618,10.686,149.520
C07153=1125.084,324.052,-79.240,-177.614,10.688,149.519
C07154=1125.079,324.300,-79.273,-177.611,10.691,149.519
C07155=1125.075,324.548,-79.307,-177.608,10.694,149.519
C07156=1125.072,324.796,-79.340,-177.605,10.696,149.519
C07157=1125.068,325.044,-79.373,-177.602,10.698,149.518
C07158=1125.064,325.291,-79.407,-177.599,10.700,149.518
C07159=1125.060,325.539,-79.440,-177.596,10.703,149.518
C07160=1125.055,325.786,-79.474,-177.592,10.705,149.518
C07161=1125.052,326.035,-79.507,-177.589,10.708,149.518
C07162=1125.048,326.282,-79.541,-177.586,10.711,149.518
C07163=1125.044,326.530,-79.574,-177.583,10.713,149.517
C07164=1125.039,326.778,-79.608,-177.579,10.716,149.517
C07165=1125.035,327.025,-79.642,-177.577,10.718,149.517
C07166=1125.032,327.273,-79.675,-177.573,10.721,149.517
C07167=1125.028,327.521,-79.708,-177.570,10.723,149.517
C07168=1125.024,327.768,-79.742,-177.567,10.726,149.517
C07169=1125.020,328.016,-79.775,-177.564,10.728,149.516
C07170=1125.015,328.263,-79.809,-177.560,10.731,149.516
C07171=1125.011,328.512,-79.843,-177.557,10.734,149.516
C07172=1125.007,328.759,-79.877,-177.554,10.736,149.516
C07173=1125.004,329.006,-79.910,-177.551,10.739,149.515
C07174=1124.999,329.254,-79.944,-177.548,10.740,149.515
C07175=1124.996,329.502,-79.978,-177.545,10.743,149.515
C07176=1124.991,329.750,-80.012,-177.542,10.745,149.515
C07177=1124.987,329.997,-80.045,-177.539,10.748,149.515
C07178=1124.984,330.246,-80.079,-177.536,10.751,149.515
C07179=1124.980,330.493,-80.113,-177.532,10.753,149.514
C07180=1124.976,330.740,-80.146,-177.529,10.756,149.514
C07181=1124.971,330.988,-80.180,-177.526,10.758,149.514
C07182=1124.968,331.236,-80.214,-177.523,10.761,149.514
C07183=1124.964,331.483,-80.248,-177.519,10.763,149.514
C07184=1124.959,331.731,-80.282,-177.516,10.766,149.513
C07185=1124.956,331.979,-80.316,-177.513,10.768,149.513
C07186=1124.952,332.226,-80.350,-177.510,10.771,149.513
C07187=1124.948,332.474,-80.383,-177.507,10.773,149.513
C07188=1124.944,332.722,-80.418,-177.503,10.776,149.513
C07189=1124.940,332.969,-80.452,-177.500,10.779,149.512
C07190=1124.936,333.217,-80.485,-177.497,10.781,149.512
C07191=1124.932,333.465,-80.520,-177.494,10.783,149.512
C07192=1124.928,333.712,-80.553,-177.491,10.785,149.512
C07193=1124.924,333.959,-80.587,-177.488,10.788,149.512
C07194=1124.920,334.208,-80.621,-177.485,10.790,149.511
C07195=1124.917,334.420,-80.651,-177.481,10.793,149.511
C07196=1124.913,334.633,-80.680,-177.479,10.795,149.511
C07197=1124.910,334.845,-80.709,-177.476,10.797,149.511
C07198=1124.907,335.058,-80.738,-177.474,10.799,149.511
C07199=1124.904,335.272,-80.768,-177.471,10.801,149.511
C07200=1124.900,335.484,-80.797,-177.468,10.804,149.510
C07201=1124.896,335.697,-80.827,-177.465,10.805,149.510
C07202=1124.893,335.910,-80.856,-177.463,10.807,149.510
C07203=1124.889,336.157,-80.890,-177.460,10.810,149.510
C07204=1124.885,336.405,-80.924,-177.456,10.812,149.510
C07205=1124.881,336.653,-80.958,-177.453,10.815,149.509
C07206=1124.877,336.901,-80.993,-177.450,10.818,149.509
C07207=1124.873,337.148,-81.027,-177.447,10.820,149.509
C07208=1124.870,337.396,-81.061,-177.443,10.822,149.509
C07209=1124.865,337.643,-81.096,-177.440,10.825,149.509
C07210=1124.862,337.890,-81.129,-177.437,10.828,149.509
C07211=1124.858,338.138,-81.164,-177.434,10.830,149.508
C07212=1124.854,338.385,-81.198,-177.431,10.833,149.508
C07213=1124.850,338.633,-81.233,-177.427,10.835,149.508
C07214=1124.845,338.881,-81.267,-177.424,10.838,149.508
C07215=1124.842,339.129,-81.302,-177.421,10.840,149.508
C07216=1124.837,339.376,-81.336,-177.418,10.843,149.507
C07217=1124.834,339.624,-81.370,-177.414,10.845,149.507
C07218=1124.830,339.871,-81.405,-177.411,10.848,149.507
C07219=1124.826,340.119,-81.440,-177.408,10.850,149.507
C07220=1124.822,340.367,-81.474,-177.405,10.852,149.507
C07221=1124.818,340.615,-81.508,-177.402,10.855,149.506
C07222=1124.814,340.862,-81.542,-177.399,10.857,149.506
C07223=1124.810,341.109,-81.578,-177.395,10.860,149.506
C07224=1124.806,341.357,-81.612,-177.393,10.862,149.506
C07225=1124.803,341.605,-81.646,-177.389,10.865,149.506
C07226=1124.798,341.852,-81.681,-177.386,10.867,149.505
C07227=1124.794,342.100,-81.716,-177.383,10.870,149.505
C07228=1124.791,342.347,-81.750,-177.379,10.872,149.505
C07229=1124.787,342.595,-81.785,-177.376,10.875,149.505
C07230=1124.782,342.842,-81.820,-177.373,10.877,149.505
C07231=1124.779,343.090,-81.854,-177.370,10.880,149.504
C07232=1124.775,343.337,-81.889,-177.366,10.882,149.504
C07233=1124.771,343.585,-81.924,-177.363,10.885,149.504
C07234=1124.767,343.833,-81.959,-177.360,10.887,149.504
C07235=1124.763,344.080,-81.993,-177.356,10.890,149.503
C07236=1124.759,344.328,-82.028,-177.354,10.892,149.503
C07237=1124.755,344.575,-82.063,-177.350,10.895,149.503
C07238=1124.751,344.823,-82.097,-177.347,10.897,149.503
C07239=1124.747,345.070,-82.132,-177.344,10.899,149.503
C07240=1124.743,345.318,-82.167,-177.341,10.901,149.502
C07241=1124.739,345.565,-82.202,-177.338,10.904,149.502
C07242=1124.735,345.813,-82.237,-177.335,10.907,149.502
C07243=1124.732,346.060,-82.272,-177.331,10.909,149.502
C07244=1124.728,346.308,-82.307,-177.328,10.912,149.502
C07245=1124.723,346.555,-82.341,-177.325,10.914,149.501
C07246=1124.720,346.803,-82.377,-177.321,10.917,149.501
C07247=1124.715,347.050,-82.411,-177.318,10.919,149.501
C07248=1124.711,347.298,-82.447,-177.315,10.921,149.501
C07249=1124.708,347.546,-82.481,-177.312,10.924,149.501
C07250=1124.704,347.792,-82.516,-177.309,10.927,149.501
C07251=1124.701,348.006,-82.547,-177.306,10.928,149.500
C07252=1124.697,348.218,-82.576,-177.303,10.931,149.500
C07253=1124.694,348.431,-82.607,-177.300,10.933,149.500
C07254=1124.691,348.643,-82.636,-177.298,10.935,149.500
C07255=1124.687,348.856,-82.667,-177.295,10.937,149.500
C07256=1124.685,349.068,-82.697,-177.292,10.939,149.499
C07257=1124.681,349.281,-82.728,-177.289,10.941,149.499
C07258=1124.677,349.494,-82.758,-177.286,10.944,149.499
C07259=1124.673,349.742,-82.793,-177.283,10.946,149.499
C07260=1124.670,349.989,-82.828,-177.279,10.949,149.499
C07261=1124.666,350.236,-82.863,-177.276,10.951,149.498
C07262=1124.662,350.484,-82.898,-177.272,10.954,149.498
C07263=1124.658,350.731,-82.933,-177.268,10.957,149.498
C07264=1124.654,350.979,-82.969,-177.265,10.960,149.498
C07265=1124.651,351.226,-83.004,-177.262,10.962,149.497
C07266=1124.646,351.474,-83.039,-177.258,10.964,149.497
C07267=1124.642,351.721,-83.074,-177.254,10.967,149.497
C07268=1124.639,351.969,-83.110,-177.251,10.970,149.497
C07269=1124.635,352.216,-83.145,-177.247,10.972,149.496
C07270=1124.631,352.463,-83.180,-177.244,10.975,149.496
C07271=1124.627,352.711,-83.215,-177.240,10.978,149.496
C07272=1124.623,352.959,-83.251,-177.236,10.980,149.495
C07273=1124.619,353.206,-83.286,-177.233,10.983,149.495
C07274=1124.615,353.453,-83.322,-177.230,10.985,149.495
C07275=1124.611,353.701,-83.358,-177.226,10.987,149.495
C07276=1124.607,353.948,-83.393,-177.222,10.990,149.494
C07277=1124.603,354.196,-83.429,-177.219,10.993,149.494
C07278=1124.600,354.443,-83.464,-177.216,10.995,149.494
C07279=1124.596,354.691,-83.500,-177.212,10.998,149.494
C07280=1124.592,354.937,-83.535,-177.209,11.000,149.494
C07281=1124.588,355.185,-83.571,-177.205,11.002,149.493
C07282=1124.585,355.432,-83.606,-177.201,11.006,149.493
C07283=1124.581,355.680,-83.642,-177.198,11.008,149.493
C07284=1124.576,355.928,-83.678,-177.195,11.011,149.493
C07285=1124.573,356.175,-83.713,-177.191,11.013,149.492
C07286=1124.569,356.423,-83.749,-177.188,11.015,149.492
C07287=1124.565,356.670,-83.784,-177.184,11.018,149.492
C07288=1124.561,356.917,-83.820,-177.181,11.020,149.491
C07289=1124.558,357.165,-83.855,-177.177,11.022,149.491
C07290=1124.553,357.412,-83.891,-177.173,11.025,149.491
C07291=1124.550,357.659,-83.928,-177.170,11.028,149.491
C07292=1124.546,357.907,-83.963,-177.167,11.030,149.490
C07293=1124.542,358.154,-83.999,-177.163,11.033,149.490
C07294=1124.538,358.402,-84.035,-177.160,11.035,149.490
C07295=1124.534,358.650,-84.070,-177.156,11.037,149.490
C07296=1124.531,358.896,-84.107,-177.153,11.040,149.489
C07297=1124.527,359.143,-84.142,-177.149,11.042,149.489
C07298=1124.522,359.391,-84.178,-177.146,11.045,149.489
C07299=1124.519,359.639,-84.214,-177.143,11.047,149.489
C07300=1124.515,359.885,-84.250,-177.140,11.049,149.488
C07301=1124.512,360.133,-84.285,-177.136,11.052,149.488
C07302=1124.507,360.381,-84.322,-177.133,11.054,149.488
C07303=1124.504,360.628,-84.358,-177.129,11.057,149.487
C07304=1124.500,360.875,-84.393,-177.126,11.059,149.487
C07305=1124.496,361.123,-84.429,-177.123,11.061,149.487
C07306=1124.493,361.370,-84.466,-177.119,11.064,149.487
C07307=1124.490,361.583,-84.497,-177.116,11.066,149.486
C07308=1124.486,361.795,-84.527,-177.113,11.068,149.486
C07309=1124.483,362.008,-84.558,-177.111,11.070,149.486
C07310=1124.479,362.220,-84.590,-177.107,11.072,149.486
C07311=1124.476,362.432,-84.621,-177.105,11.074,149.486
C07312=1124.473,362.645,-84.652,-177.101,11.076,149.485
C07313=1124.470,362.858,-84.683,-177.099,11.078,149.485
C07314=1124.466,363.070,-84.714,-177.095,11.081,149.485
C07315=1124.462,363.317,-84.750,-177.093,11.082,149.485
C07316=1124.459,363.564,-84.786,-177.089,11.085,149.484
C07317=1124.455,363.812,-84.822,-177.086,11.087,149.484
C07318=1124.451,364.059,-84.858,-177.082,11.089,149.484
